// POUs/IO/AnalogInELMSingleSampleDINT
// AnalogIn FB to read and scale a single DINT (24bit) sample input from ELMxxxx terminal
// Set bit 3 (Options.3) to true to enable scaling based on +/-7812500 instead of legacy range values +/-838860x
FUNCTION_BLOCK AnalogInELMSingleSampleDINT EXTENDS AnalogInELMBase
VAR_INPUT
	Offset													:	LREAL := 0.0;

END_VAR                 									
VAR                                     	            	
END_VAR                                 	            	
VAR_OUTPUT                              	            	                                       	
	Q														:	LREAL;	//scaled result value
	In											AT  %I* 	: 	DINT; 	//Hardware Input 
END_VAR                                 	
VAR                                   	
END_VAR

(* Read single DINT sample value from ELM terminal and scale to user units									*)
(************************************************************************************************************)

(* evaluate statusword **************************************************************************************)
	SUPER^();
	
(* Scaling ******************************************************************)
	IF MaxValue <> MinValue 
	THEN	
		IF NOT Options.3
		THEN
			Q 	 											:= Offset + Scale(TO_LREAL(In) , -8388608.0, 8388607.0, MinValue , MaxValue);
		ELSE
			Q 	 											:= Offset + Scale(TO_LREAL(In), -7812500.0, 7812500.0, MinValue , MaxValue);
		END_IF	
		IF NoOfDigits > 0
		THEN
			Q												:= TO_FMLREAL(Q,NoOfDigits);
		END_IF
	
	ELSIF NoOfDigits > 0 (* Bsp PT100 *)
	THEN
		Q													:= Offset + TO_FMLREAL(In,NoOfDigits);
		
	ELSE  													
		Q 													:= 0.0;
	END_IF

	IF 	Error AND OutOnError <> 0.000000000000000001
	THEN
		Q													:= OutOnError;
	END_IF
(**********************************************************************************************************************)

METHOD FB_init : BOOL
VAR_INPUT
	bInitRetains : BOOL; // if TRUE, the retain variables are initialized (warm start / cold start)
	bInCopyCode : BOOL;  // if TRUE, the instance afterwards gets moved into the copy code (online change)
END_VAR
IF NOT bInCopyCode THEN
	NoOfDigits 							:= 2;
END_IF
END_METHOD

PROPERTY PUBLIC optEnableScaleExtRangeMode : bool
GET
optEnableScaleExtRangeMode := Options.3;
END_GET
SET
Options.3 := optEnableScaleExtRangeMode;
END_SET
END_PROPERTY

END_FUNCTION_BLOCK

// POUs/IO/AnalogInELMSingleSampleREAL
// AnalogIn FB to read and scale a single REAL sample input from ELMxxxx terminal
// Set bit 3 (Options.3) to true to enable scaling based on +/-7812500 instead of legacy range values +/-838860x
// NoOfDigits per default set to 3... 
FUNCTION_BLOCK AnalogInELMSingleSampleREAL EXTENDS AnalogInELMBase
VAR_INPUT
	Offset													:	LREAL := 0.0;
END_VAR                 									
VAR                                     	            	
END_VAR                                 	            	
VAR_OUTPUT                              	            	                                       	
	Q														:	LREAL;	//scaled result value
	In											AT  %I* 	: 	REAL; 	//Hardware Input 
END_VAR                                 	
VAR                                     	
END_VAR

(* Read single REAL sample value from ELM terminal and scale to user units									*)
(************************************************************************************************************)

(* evaluate statusword **************************************************************************************)
	SUPER^();
	
(* Scaling ******************************************************************)
	IF MaxValue <> MinValue 
	THEN			
		IF NOT Options.3
		THEN
			Q 	 											:= Offset + Scale(TO_LREAL(In), -8388608.0, 8388607.0, MinValue , MaxValue);
		ELSE
			Q 	 											:= Offset + Scale(TO_LREAL(In),  -7812500.0, 7812500.0, MinValue , MaxValue);		
		END_IF	
		
		IF NoOfDigits > 0
		THEN
			Q												:= TO_FMLREAL(Q,NoOfDigits);
		END_IF
	
	ELSIF NoOfDigits > 0 (* Bsp PT100 *)
	THEN
		Q													:= Offset + TO_FMLREAL(In,NoOfDigits);
		
	ELSE  													
		Q 													:= 0.0;
	END_IF


(**********************************************************************************************************************)

METHOD FB_init : BOOL
VAR_INPUT
	bInitRetains : BOOL; // if TRUE, the retain variables are initialized (warm start / cold start)
	bInCopyCode : BOOL;  // if TRUE, the instance afterwards gets moved into the copy code (online change)
END_VAR
IF NOT bInCopyCode THEN
	NoOfDigits 							:= 3;
END_IF
END_METHOD

PROPERTY PUBLIC optEnableScaleExtRangeMode : bool
GET
optEnableScaleExtRangeMode := Options.3;
END_GET
SET
Options.3 := optEnableScaleExtRangeMode;
END_SET
END_PROPERTY

END_FUNCTION_BLOCK

// POUs/IO/BlowOffSensors
{attribute 'no_check'}
//FB generates a pulse "Pulse" time based signal on every bit at Q (DWORD) for a certain lenght
//The sequecne will starts based on the seletcted time of interval if Enable is TRUE
//The FB can be used to activate air blow valves on by one to clean sensors in a dusty environment
FUNCTION_BLOCK BlowOffSensors
VAR_INPUT
	Enable													:	BOOL;			//FB will be processed as long as enable is TRUE
	StartManual												:	BOOL;			//starts FB without interval
	Interval												:	TIME := T#60M; 	//Blow of autostart interval
	Lenght													:	TIME := T#4S; 	//Duration of pulsing
	Pulse													:	TIME := T#500MS; //On/Off pulse duration
END_VAR                 									
VAR_OUTPUT              									
	Aktiv													:	BOOL;			//Busy is TRUE at the rising edge of Enable and stays TRUE as long as the FB is performing any action.  
{attribute 'displaymode':='binary'}    
	Q														:	DWORD := 0;		//Each bit will be set and reset based on the settings one by one 
END_VAR                 									
VAR                     									
	state													:	INT := 0;
	i														:	SINT ;
	TON_Interval											:	TON;
	TON_Lenght		 										: 	TON;
	TOF_Pulse	 											:	TOF;
END_VAR

(* Abblastaktgenerator					*)
(***************************************)

(* Intervalzeit ***********************************************************************)
IF Enable 
THEN
	CASE state OF
	0:
		TON_Interval(IN := FALSE);
		state 												:= 10;
		i 													:= -1;

	1:
		Aktiv := FALSE;
		TON_Interval(IN := Interval <> T#0MS , PT := Interval);
		IF TON_Interval.Q
			OR StartManual
		THEN
			TON_Interval(IN := FALSE);
			
			state 											:= 10;
			Aktiv 											:= TRUE;
			i 												:= -1;
		END_IF

	10:
		i := i + 1;
		IF i > 31 THEN
			state 											:= 1;
		ELSE
			TON_Lenght(IN := FALSE);
			TOF_Pulse(IN := FALSE);
			
			Q		 										:= 0;
			state 											:= 11;
		END_IF                  							

	11:
		TON_Lenght(IN := TRUE, PT := Lenght);

		IF 	TON_Lenght.Q
			AND Q = 0
		THEN
			state 											:= 10;
		ELSE
			IF 	NOT TOF_Pulse.Q 
				AND Q <> 0 
			THEN
				TOF_Pulse(IN:=TRUE  , PT:= Pulse);
				Q		 									:= 0;
			ELSIF NOT TOF_Pulse.Q 
				AND Q = 0 
			THEN
				TOF_Pulse(IN:= TRUE , PT:= Pulse) ;
				Q		 									:= SETBIT32(Q,i);
			END_IF
			(* Work Timer *)
			TOF_Pulse(IN:=FALSE);
		END_IF

	END_CASE
ELSE
	Aktiv 													:= FALSE;
	state 													:= 0;
	Q														:= 0;
END_IF

(**********************************************************************************************************)

END_FUNCTION_BLOCK

// POUs/TimeHelper/Pulse
{attribute 'no_check'}
//Generates a pulse signal 
FUNCTION_BLOCK Pulse
VAR_INPUT
	IN														: BOOL; //Start pulse generator
	PT_ON													: TIME; //Time pulse on	
	PT_OFF													: TIME; //Time pulse off 
END_VAR             										
VAR_OUTPUT          										
	Q														: BOOL; 
	RT														: BOOL; 
	FT														: BOOL;
END_VAR             										
VAR                 	
	TON_PULSE												: TON;
END_VAR

	(* Pulse generator																*)
	(********************************************************************************)

(* Reset flag *)
RT := FT													:= FALSE;
(* logic *)
IF 	Q AND(TON_PULSE.Q OR NOT IN)
THEN
	TON_PULSE(IN:=FALSE  , PT:= PT_OFF);
	FT 														:= Q;
	Q 														:= FALSE;
ELSIF NOT Q AND TON_PULSE.Q
	OR_ELSE In AND NOT TON_PULSE.IN 
THEN
	RT 														:= NOT Q;
	TON_PULSE(IN:= FALSE , PT:= PT_ON) ;
	Q 														:= TRUE;
END_IF

//Run timer
TON_PULSE(IN:=IN);

(***********************************************************************************************************************)

END_FUNCTION_BLOCK

// POUs/IO/Button
{attribute 'no_check'}
FUNCTION_BLOCK Button 
VAR_INPUT
	Enable													:	BOOL := TRUE;	//FB will be processed as long as enable is TRUE 
	RstTGL													:	BOOL := FALSE; 	//resets the Toggle signal
	SetTGL													:	BOOL := FALSE;	//sets the Toggle signal
	Force													:	BOOL := FALSE; 	//simulates Input signal
	Invert													:	BOOL := FALSE; 	//inverts the Hardware Input
	LED												AT  %Q*	:	BOOL;			//LED/Light hardware output
END_VAR         									
VAR_OUTPUT
	Q														:	BOOL;	//direct signal
	Q_RT													:	BOOL;	//R_Trig signal of delay Q
	Q_FT													:	BOOL;	//F_Trig signal of delay Q
	Q_TGL													:	BOOL;	//Toggle -> use flag Q_RT
	In												AT  %I*	:	BOOL; 	//Hardware Input
END_VAR
VAR
	Mem														:	BOOL;
END_VAR

(* Taster mit Togglefunktion V1.0						*)
(********************************************************)

(********************************************************)
Mem															:= Q;
Q 															:= ((In OR Force) XOR Invert) AND Enable;
Q_RT 														:= NOT Mem AND Q;
Q_FT														:= Mem AND NOT Q;
Q_TGL 														:= (Q_RT XOR Q_TGL);
(********************************************************)

METHOD PUBLIC setDisable : BOOL
VAR_INPUT
END_VAR
Enable 														:= FALSE;
setDisable													:= TRUE;
END_METHOD

METHOD PUBLIC setEnable : bool
VAR_INPUT
END_VAR
Enable 														:= TRUE;
setEnable													:= TRUE;
END_METHOD

METHOD PUBLIC setLedOFF : bool
VAR_INPUT
END_VAR
LED 														:= FALSE;
setLEDOff													:= TRUE;
END_METHOD

METHOD PUBLIC setLedON : booL
VAR_INPUT
END_VAR
LED 														:= TRUE;
setLedON													:= TRUE;
END_METHOD

METHOD PUBLIC TGL : booL //Return value = Q_TGL status
VAR_INPUT
END_VAR
TGL := Q_TGL 														:= NOT Q_TGL;
END_METHOD

METHOD PUBLIC TglOff : booL
VAR_INPUT
END_VAR
Q_TGL 														:= FALSE;
TglOFF														:= TRUE;
END_METHOD

METHOD PUBLIC TglOn : bool
VAR_INPUT
END_VAR
Q_TGL 														:= TRUE;
TglON														:= TRUE;
END_METHOD

END_FUNCTION_BLOCK

// POUs/IO/ButtonExt
{attribute 'no_check'}
//Button with delay function 
FUNCTION_BLOCK ButtonExt EXTENDS Button
VAR_INPUT
	PT_ON													:	TIME := T#0MS; 	//Delay for Q, Q_RT (TGL) and Q_FT
END_VAR
VAR_OUTPUT
	Q_DIRECT												:	BOOL; 	//Direct signal - undelayed
END_VAR
VAR
	TON														:	TON;
END_VAR

(* Button with toggle-function and on-delay		V1.5	*)
(********************************************************)

(********************************************************)
TON(IN := ((In OR Force) XOR Invert) AND Enable, PT := PT_ON);
Q_DIRECT 													:= TON.IN;
IF NOT Q    												
THEN        												
	Q 														:= TON.Q;
	Q_RT 													:= Q;
	Q_FT 													:= FALSE;
ELSE        												
	Q 														:= TON.IN;
	Q_RT 													:= FALSE;
	Q_FT 													:= NOT Q;
END_IF      	

Q_TGL := NOT RstTGL AND (Q_RT XOR Q_TGL OR SetTGL) ;

(********************************************************)

END_FUNCTION_BLOCK

// POUs/IO/InOut
{attribute 'no_check'}
FUNCTION_BLOCK InOut 
VAR_INPUT
	Q												AT  %Q*	:	BOOL; //Link to hardware output
END_VAR             								
VAR_OUTPUT          								
	In												AT  %I*	:	BOOL; //Link to hardware input
END_VAR
VAR
END_VAR

;

END_FUNCTION_BLOCK

// POUs/IO/InOutExt
{attribute 'no_check'}
FUNCTION_BLOCK InOutExt EXTENDS InOut IMPLEMENTS I_ActuatorOnOff
VAR_INPUT
	ResetTrig												:	BOOL;	//Resets error with rising edge
	Invert													:	BOOL ;			//Inverts the logic of varibale In (AT  %I*)
	PT_Timeout												:	TIME := T#3S;  	//Time value until Timeout of process (Error)
END_VAR                     				
VAR_OUTPUT                  				
	Busy													:	BOOL;			//Busy is TRUE at the rising edge of Execute and FALSE when one of the outputs Done, Aborted, or Error is set 
	ErrorOn													:	BOOL;			//Timeout error waiting for IN changing to TRUE
	ErrorOff												:	BOOL;			//Timeout error waiting for IN changing to FALSE
	Done													:	BOOL;			//The Done output is set when the commanded action has been completed successfully 
	Status													:	BYTE;			//8 different query Options (conditions see below)
END_VAR                     	
VAR                         	
	tonRM													:	ton;			
END_VAR

(* Actuator with feedback								*)
(********************************************************)

(********************************************************)
	IF Q 
	THEN
		SwitchOn();
	ELSE
		SwitchOff();
	END_IF
	_runtimeChk();
	_writeStatus();

(********************************************************)

METHOD PROTECTED _runtimeChk : BOOL
VAR_INPUT
END_VAR
	tonRM(
		IN	:= Busy AND NOT ResetTrig,  
		PT 	:= PT_Timeout,
		Q	=> );
		
	ErrorOff 												:= tonRM.Q AND NOT Q;
	ErrorOn 												:= tonRM.Q AND Q;

	_runtimeChk									:= TRUE;
END_METHOD

METHOD PROTECTED _writeStatus : BOOL
VAR_INPUT
END_VAR
	Status.0 												:= NOT Q;
	Status.1 												:= Q;
	Status.2 												:= NOT (In XOR Invert);
	Status.3 												:= In XOR Invert;
	Status.4 												:= NOT ErrorOff;
	Status.5 												:= NOT ErrorOn;
	Status.6 												:= NOT Status.7;
	Status.7 												:= ErrorOff OR ErrorOn;
	
	(* Result *)
	_writeStatus											:= TRUE;
END_METHOD

METHOD PUBLIC enable : BOOL //Result value = TRUE if successful executed (
VAR_INPUT 
	IN								: BOOL; //TRUE = ON/FALSE = OFF	
END_VAR
IF IN
THEN
	enable							:= switchOn();
ELSE
	enable							:= switchOff();
END_IF
END_METHOD

{attribute 'monitoring' := 'call'}
PROPERTY public inError : BOOL
GET
inError := ErrorON or ErrorOff;
END_GET
END_PROPERTY

{attribute 'monitoring' := 'call'}
PROPERTY public isBusy : bool
GET
isBusy := Busy;
END_GET
END_PROPERTY

{attribute 'monitoring' := 'call'}
PROPERTY public isOff : BOOL
GET
isOff := not Q;
END_GET
END_PROPERTY

{attribute 'monitoring' := 'call'}
PROPERTY public isOn : BOOL
GET
isOn := Q;
END_GET
END_PROPERTY

{attribute 'monitoring' := 'call'}
PROPERTY Public noFeed : BOOL
GET
noFeed := FALSE;
END_GET
END_PROPERTY

{attribute 'monitoring' := 'call'}
PROPERTY Public ok : bool
GET
ok := Q and Done or not Q and not Done;
END_GET
END_PROPERTY

METHOD PUBLIC reset : Bool
VAR_INPUT
END_VAR
tonRM(IN := FALSE);
reset := TRUE;
END_METHOD

METHOD public switchOff : BOOL
VAR_INPUT
END_VAR
	
	Q														:= FALSE;
	Done													:= NOT (In XOR Invert);
	Busy													:= NOT Done;
	switchOff												:= Done;
END_METHOD

METHOD public switchOn : BOOL
VAR_INPUT
END_VAR
	Q														:= TRUE;
	Done													:= (In XOR Invert);
	Busy													:= NOT Done;
	switchOn												:= Done;
END_METHOD

END_FUNCTION_BLOCK

// POUs/IpcDiag/MDP/InfoModuls/MDP_CPU
{attribute 'no_check'}
//Wrapper for available MDP_xxxx FBs of the lib, based on Beckhoff MDP - invalid values are reported via EventLogger 
//based on Tc2_MDP.lib - please see Beckhoff documentation for further information about Tc2_MDP.lib (IPC diagnostics)
FUNCTION_BLOCK MDP_CPU  EXTENDS FbBase
VAR_OUTPUT CONSTANT
	MIN_CPU													:	INT := 1;
	MAX_CPU													:	INT := 8;
END_VAR                 									
VAR_INPUT               									
	AmsNetId												: 	T_AmsNetId := '';				//AmsNetId as text
	Timeout													:	TIME := DEFAULT_ADS_TIMEOUT;	//Ads timeout
END_VAR                 									
VAR_OUTPUT              									
	Frequency												:  ARRAY[MIN_CPU..MAX_CPU] OF	UDINT;	//current CPU frequency
	Usage													:	ARRAY[MIN_CPU..MAX_CPU] OF	UINT;	//current CPU usage in %
	Temperature												:	ARRAY[MIN_CPU..MAX_CPU] OF	INT;	//current CPU temperature in °C
	AverageFrequency 										:	UDINT;		//average CPU frequency
	AverageUsage	 										:	UINT;		//average CPU usage in %
	AverageTemperature										:	INT;		//average CPU temperature in °C
	Count													:	INT; 		//number of CPUs
	ErrorGrp												:	E_MDP_ErrGroup := eMDP_Err_NoError;
END_VAR
VAR
	idx														:	INT := 1;
	MDP_ScanModules											:	FB_MDP_ScanModules := ( nModuleType 	:= eMDP_ModT_CPU , iModIdx		:= 0);
	MDP_Read												: 	FB_MDP_ReadModuleContent;
	SplitErrorId											:	FB_MDP_SplitErrorID;
	DstBuf													:	ARRAY[0..13] OF BYTE;
END_VAR

(* Read CPU Information 						V1.0		*)
(************************************************************)

(* Start Read ***********************************************)
	IF Execute
		AND state = 0
	THEN
		MEMSET(ADR(Frequency),0,SIZEOF(Frequency));
		MEMSET(ADR(Usage),0,SIZEOF(Usage));
		MEMSET(ADR(Temperature),0,SIZEOF(Temperature));
		AverageFrequency									:= 0;
		AverageUsage										:= 0;
		AverageTemperature									:= 0;
		Count												:= 0;
		Busy												:= TRUE;
		Done												:= FALSE;
		Error												:= FALSE;
		ErrorId												:= 0;
		ErrorGrp											:= eMDP_Err_NoError;
		MDP_Read(bExecute := FALSE);
		MDP_ScanModules(
			bExecute		:= FALSE,
			nModuleType		:= eMDP_ModT_CPU,
			iModIdx			:= 0,
			tTimeout		:= timeout,
			sAmsNetId		:= AmsNetId,
			bBusy			=> ,
			bError			=> ,
			nErrID			=> ,
			nDynModuleId	=> ,
			iModuleTypeCount=> ,
			iModuleCount	=> );
			
		MDP_ScanModules(bExecute		:= TRUE);		
		state												:= 1 ;
		
	ELSIF NOT Execute
		AND State = 99
	THEN
		state												:= 0;
		Busy												:= FALSE;
		Done												:= FALSE;
		Error												:= FALSE;
		ErrorId												:= 0;
		ErrorGrp											:= eMDP_Err_NoError;
	END_IF


	CASE state OF
	0:
		;
	1:
		MDP_ScanModules();
		IF NOT MDP_ScanModules.bBusy
		THEN
			IF MDP_ScanModules.bError
			THEN
				Busy										:= FALSE;
				Error										:= TRUE;
				SplitErrorId(
					nErrID		:= MDP_ScanModules.nErrID,
					eErrGroup	=> ErrorGrp ,
					nErrCode	=> ErrorId);
				state										:= 99;
				MDP_ScanModules(bExecute := FALSE);
			ELSE
				Count										:= MDP_ScanModules.iModuleTypeCount;
				MDP_Read.stMDP_DynAddr.nArea				:= 16#8;
				MDP_Read.stMDP_DynAddr.nModuleId			:= MDP_ScanModules.nDynModuleId;
				MDP_Read.stMDP_DynAddr.nSubIdx				:= 0;
				MDP_Read.stMDP_DynAddr.nTableId				:= 1;
				MDP_Read(bExecute := FALSE);
				idx											:= 1;
				IF Count = 0
				THEN
					Busy									:= FALSE;
					Error									:= TRUE;
					ErrorId									:= MDP_Read.nErrID;
					state									:= 99;
				ELSE
					MDP_Read(
						bExecute		:= TRUE,
						stMDP_DynAddr	:= ,
						iSubIdxCount	:= 4,
						pDstBuf			:= ADR(DstBuf),
						cbDstBufLen		:= SIZEOF(DstBuf),
						tTimeout		:= timeout,
						sAmsNetId		:= AmsNetId,
						bBusy			=> ,
						bError			=> ,
						nErrID			=> ,
						iErrPos			=> ,
						arrStartIdx		=> );
					state									:= 2;
				END_IF
			END_IF

		END_IF

	2:
		MDP_Read( pDstBuf := ADR(DstBuf), cbDstBufLen := SIZEOF(DstBuf));
		
		IF NOT MDP_Read.bBusy
		THEN
			IF MDP_Read.bError AND MDP_Read.iErrPos <> 4 AND MDP_Read.bExecute
			THEN
				Busy										:= FALSE;
				Error										:= TRUE;
				SplitErrorId(
					nErrID		:= MDP_Read.nErrID,
					eErrGroup	=> ErrorGrp ,
					nErrCode	=> ErrorId);
				state										:= 99;
				MDP_Read(bExecute := FALSE);
			ELSE
				(* copy freq *)
				IF MDP_Read.arrStartIdx[1] >= 0
				THEN
					MEMCPY( ADR(Frequency[idx]) , ADR(DstBuf[MDP_Read.arrStartIdx[1]]) , SIZEOF(Frequency[idx]) );
				END_IF
				(* copy usage *)
				IF MDP_Read.arrStartIdx[2] <> 0
				THEN
					MEMCPY(ADR(Usage[idx]) , ADR(DstBuf[MDP_Read.arrStartIdx[2]]) , SIZEOF(Usage[idx]) );
				END_IF
				(* copy temp in availible *)
				IF MDP_Read.arrStartIdx[3] <> 0
				THEN
					MEMCPY(ADR(Temperature[idx]) , ADR(DstBuf[MDP_Read.arrStartIdx[3]]) , SIZEOF(Temperature[idx]) ) ;
				END_IF

				MDP_Read(bExecute := FALSE);
				MDP_Read.stMDP_DynAddr.nModuleId := MDP_Read.stMDP_DynAddr.nModuleId + 1;
				
				idx 										:= idx + 1;
				IF idx > Count AND Count > 0
				THEN
					FOR idx := 1 TO Count
					DO
						AverageFrequency 					:= AverageFrequency + Frequency[idx];
						AverageUsage 						:= AverageUsage + Usage[idx];
						AverageTemperature 					:= AverageTemperature + Temperature[idx];
					END_FOR                         		
                                                    		
					AverageFrequency						:= AverageFrequency / INT_TO_UDINT(Count);
					AverageUsage							:= AverageUsage / INT_TO_UINT(Count);
					AverageTemperature						:=	AverageTemperature / INT_TO_SINT(Count);
                                                        	
					Busy									:= FALSE;
					Done									:= TRUE;
					state									:= 99;
				ELSE
					MDP_Read(bExecute := TRUE);
				END_IF
			END_IF
		END_IF

	99: ;

	ELSE
		;
	END_CASE

	(* reset state for next start *)
	IF NOT Execute
		AND state = 99
	THEN
		state												:= 0;
	END_IF

(****************************************************************************************************)

END_FUNCTION_BLOCK

// POUs/IpcDiag/MDP/InfoModuls/MDP_Fan
{attribute 'no_check'}
FUNCTION_BLOCK MDP_Fan EXTENDS FbBase
VAR_OUTPUT CONSTANT
	MIN_FAN													:	INT := 1;
	MAX_FAN													:	INT := 4;
END_VAR                     								
VAR_INPUT                   								
	AmsNetId												: 	T_AmsNetId := '';					//AmsNetId as text
	Timeout													:	TIME := DEFAULT_ADS_TIMEOUT;		//Ads timeout
END_VAR                     								
VAR_OUTPUT                  								
	Speed													:  ARRAY[MIN_FAN..MAX_FAN] OF	INT;	//current fan speed
	Count													:	INT; 	//number of CPUs
	ErrorGrp												:	E_MDP_ErrGroup := eMDP_Err_NoError;
END_VAR                     								
VAR                         								
	idx														:	INT := 1;
	MDP_ScanModules											:	FB_MDP_ScanModules := ( nModuleType 	:= eMDP_ModT_FAN , iModIdx		:= 0);
	MDP_Read												: 	FB_MDP_Read;
	SplitErrorId											:	FB_MDP_SplitErrorID;
	DstBuf													:	ARRAY[0..4] OF BYTE;
END_VAR

(* Read FAN Information 					V1.0	*)
(****************************************************)

(* Start Read *******************************************************)
	IF Execute
		AND state = 0
	THEN
		MEMSET(ADR(Speed),0,SIZEOF(Speed));
		Count												:= 0;
		Busy												:= TRUE;
		Done												:= FALSE;
		Error												:= FALSE;
		ErrorId												:= 0;
		ErrorGrp											:= eMDP_Err_NoError;
		MDP_Read(bExecute := FALSE);
		MDP_ScanModules(
			bExecute		:= FALSE,
			nModuleType		:= eMDP_ModT_FAN,
			iModIdx			:= 0,
			tTimeout		:= timeout,
			sAmsNetId		:= AmsNetId,
			bBusy			=> ,
			bError			=> ,
			nErrID			=> ,
			nDynModuleId	=> ,
			iModuleTypeCount=> ,
			iModuleCount	=> );
			
		MDP_ScanModules(bExecute		:= TRUE);		
		state												:= 1;
		
	ELSIF NOT Execute
		AND State = 99
	THEN
		state												:= 0;
		Busy												:= FALSE;
		Done												:= FALSE;
		Error												:= FALSE;
		ErrorId												:= 0;
		ErrorGrp											:= eMDP_Err_NoError;
	END_IF


	CASE state OF
	0:
		;

	1:
		MDP_ScanModules();
		IF NOT MDP_ScanModules.bBusy
		THEN
			IF MDP_ScanModules.bError
			THEN
				Busy										:= FALSE;
				Error										:= TRUE;
				SplitErrorId(
					nErrID		:= MDP_ScanModules.nErrID,
					eErrGroup	=> ErrorGrp ,
					nErrCode		=> ErrorId);
				state										:= 99;
				MDP_ScanModules(bExecute := FALSE);
			ELSE
				Count										:= MDP_ScanModules.iModuleTypeCount;
				MDP_Read(bExecute := FALSE);
				MDP_Read.stMDP_DynAddr.nArea				:= 16#8;
				MDP_Read.stMDP_DynAddr.nModuleId			:= MDP_ScanModules.nDynModuleId;
				MDP_Read.stMDP_DynAddr.nTableId				:= 1;
				MDP_Read.stMDP_DynAddr.nSubIdx				:= 1;
				
				MDP_Read(
					stMDP_DynAddr	:= ,		(* address to request subindex Count of AdressList *)
					pDstBuf			:= ADR(DstBuf),
					cbDstBufLen		:= SIZEOF(DstBuf),
					bExecute		:= TRUE,
					tTimeout		:= Timeout,
					sAmsNetId		:= AmsNetId,
					bBusy			=> ,
					bError			=> ,
					nErrId			=> );
				idx											:= 1;
				state										:= 2;
			END_IF

		END_IF

	2:
		MDP_Read( pDstBuf	:= ADR(DstBuf), cbDstBufLen := SIZEOF(DstBuf));
		IF NOT MDP_Read.bBusy
		THEN
			IF MDP_Read.bError AND MDP_Read.bExecute
			THEN
				Busy										:= FALSE;
				Error										:= TRUE;
				SplitErrorId(
					nErrID		:= MDP_Read.nErrID,
					eErrGroup	=> ErrorGrp ,
					nErrCode	=> ErrorId);
				state										:= 99;
				MDP_Read(bExecute := FALSE);
			ELSE
				MDP_Read(bExecute := FALSE);
				MEMCPY(ADR(Speed[idx]), ADR(DstBuf), SIZEOF(Speed[idx]));
				IF idx < Count
				THEN
					MDP_Read.stMDP_DynAddr.nModuleId		:= MDP_Read.stMDP_DynAddr.nModuleId + 1;
					idx 									:= idx + 1;
				ELSE                                    	
					Busy									:= FALSE;
					Done									:= TRUE;
					state									:= 99;
				END_IF

				MDP_Read(
					stMDP_DynAddr	:= ,(* address to request subindex Count of AdressList *)
					pDstBuf			:= ADR(DstBuf),
					cbDstBufLen		:= SIZEOF(DstBuf),
					bExecute		:= NOT MDP_Read.bBusy AND state = 2,
					tTimeout		:= Timeout,
					sAmsNetId		:= AmsNetId,
					bBusy			=> ,
					bError			=> ,
					nErrId			=> );
			END_IF
		END_IF

	99: ;

	ELSE
		;
	END_CASE


	(* reset state for next start *)
	IF NOT Execute
		AND state = 99
	THEN
		state												:= 0;
	END_IF

(****************************************************************************************************)

END_FUNCTION_BLOCK

// POUs/IpcDiag/MDP/InfoModuls/MDP_Mainboard
{attribute 'no_check'}
FUNCTION_BLOCK MDP_Mainboard  EXTENDS FbBase
VAR_OUTPUT CONSTANT
	MIN_VOLTAGE												:	INT := 1;
	MAX_VOLTAGE												:	INT := 20;

(* Voltage Location *)
 	VLOC_UNKNOWN											:	INT := 0;
	VLOC_OTHER												:	INT := 1;
 	VLOC_PROCESSOR											:	INT := 2;
 	VLOC_DISK												:	INT := 3;
 	VLOC_SYSTEM_MANAGEMENT_MODULE							:	INT := 4;
 	VLOC_MOTHERBOARD										:	INT := 5;
 	VLOC_MEMORY_MODULE										:	INT := 6;
 	VLOC_POWER_SUPPLY										:	INT := 7;
 	VLOC_ADDIN_CARD											:	INT := 8;
 	VLOC_FRONT_PANEL_BOARD									:	INT := 9;
 	VLOC_BACK_PANEL_BOARD									:	INT := 10;
 	VLOC_PERIPHERIE											:	INT := 11;
 	VLOC_CHASSIS											:	INT := 12;
 	VLOC_BATTERY											:	INT := 13;
 	VLOC_UPS												:	INT := 14;
	VLOC_GRAFFIC_BOARD										:	INT := 15;
 	VLOC_SUPERIO											:	INT := 16;
	VLOC_CHIPSET											:	INT := 17;
END_VAR                             						
VAR_INPUT                           						
	AmsNetId												: 	T_AmsNetId := '';				//AmsNetId as text
	Timeout													:	TIME := DEFAULT_ADS_TIMEOUT;	//Ads timeout
END_VAR
VAR_OUTPUT
	MB_Type													:	STRING(20);	//Type of Mainboard
	SerielNo												:	STRING(20);	//Serial number of Mainboard
	ProdDate												:	STRING(20);	//Production date of Mainboard
	BootCount												:	UDINT;		//total number of boots
	OpTime													:	UDINT; 		//Operating Time
	MinBoardTemp											:	DINT;		//minimum board temperature
	MaxBoardTemp											:	DINT;		//maximum board temperature
	MinInputVolt											:	DINT;		//minimum board input voltage
	MaxInputVolt											:	DINT;		//maximum board input voltage
	MB_Temp													:	INT;		//current board temperature
	IPC_SerielNo											:	STRING(20);	//industrial PC serial number
                        									
	VoltLocation											:  	ARRAY[MIN_VOLTAGE..MAX_VOLTAGE] OF INT;	//voltage location
	VoltageValue											:	ARRAY[MIN_VOLTAGE..MAX_VOLTAGE] OF INT;	//voltage value
	VoltageNominal											:	ARRAY[MIN_VOLTAGE..MAX_VOLTAGE] OF INT;	//nominal voltage
	VoltCount												:	INT; 		//number of measuring points
	ErrorGrp												:	E_MDP_ErrGroup := eMDP_Err_NoError;

END_VAR                 									
VAR                     									
	idx														:	INT := 1;
	MDP_ScanModules											:	FB_MDP_ScanModules := ( nModuleType 	:= eMDP_ModT_Mainboard , iModIdx		:= 0);
	MDP_Read												: 	FB_MDP_Read;
	SplitErrorId											:	FB_MDP_SplitErrorID;
	DstBuf													:	ARRAY[0..21] OF BYTE;
END_VAR

(* Read Mainboard Information 				V1.0	*)
(****************************************************)

(* Start Read *******************************************************)
	IF Execute
		AND state = 0
	THEN
		MB_Type												:= '';
		SerielNo											:= '';
		ProdDate											:= '';
		BootCount											:= 0;
		OpTime												:= 0;
		MinBoardTemp										:= 0;
		MaxBoardTemp										:= 0;
		MinInputVolt										:= 0;
		MaxInputVolt										:= 0;
		MB_Temp												:= 0;
		MEMSET(ADR(VoltLocation),0,SIZEOF(VoltLocation));
		MEMSET(ADR(VoltageValue),0,SIZEOF(VoltageValue));
		MEMSET(ADR(VoltageNominal),0,SIZEOF(VoltageNominal));
		VoltCount											:= 0;

		Busy												:= TRUE;
		Done												:= FALSE;
		Error												:= FALSE;
		ErrorId												:= 0;
		ErrorGrp											:= eMDP_Err_NoError;
		MDP_Read(bExecute := FALSE);
		MDP_ScanModules(
			bExecute			:= FALSE,
			nModuleType			:= eMDP_ModT_Mainboard,
			iModIdx				:= 0,
			tTimeout			:= timeout,
			sAmsNetId			:= AmsNetId,
			bBusy				=> ,
			bError				=> ,
			nErrID				=> ,
			nDynModuleId		=> ,
			iModuleTypeCount	=> ,
			iModuleCount		=> );

		MDP_ScanModules(bExecute:= TRUE);	
		state												:= 1;
		
	ELSIF NOT Execute
		AND State = 99
	THEN
		state												:= 0;
		Busy												:= FALSE;
		Done												:= FALSE;
		Error												:= FALSE;
		ErrorId												:= 0;
		ErrorGrp											:= eMDP_Err_NoError;
	END_IF


	CASE state OF
	0:
		;

	1:
		MDP_ScanModules();
		IF NOT MDP_ScanModules.bBusy
		THEN
			IF MDP_ScanModules.bError
			THEN
				Busy										:= FALSE;
				Error										:= TRUE;
				SplitErrorId(
					nErrID		:= MDP_ScanModules.nErrID,
					eErrGroup	=> ErrorGrp ,
					nErrCode	=> ErrorId);
				state										:= 99;
				MDP_ScanModules(bExecute := FALSE);
			ELSE
				MDP_Read(bExecute := FALSE);
				MDP_Read.stMDP_DynAddr.nArea				:= 16#8;
				MDP_Read.stMDP_DynAddr.nModuleId			:= MDP_ScanModules.nDynModuleId;
				MDP_Read.stMDP_DynAddr.nTableId				:= 1;
				MDP_Read.stMDP_DynAddr.nSubIdx				:= 0;
				idx											:= 1;
				state										:= 2;
			END_IF                                  		

		END_IF

	2:
		MDP_Read( pDstBuf	:= ADR(DstBuf), cbDstBufLen := SIZEOF(DstBuf));
		IF NOT MDP_Read.bBusy
		THEN
			IF MDP_Read.bError AND MDP_Read.bExecute
			THEN
				Busy										:= FALSE;
				Error										:= TRUE;
				SplitErrorId(
					nErrID		:= MDP_Read.nErrID,
					eErrGroup	=> ErrorGrp ,
					nErrCode	=> ErrorId);
				state										:= 99;
				MDP_Read(bExecute := FALSE);
			ELSE
				MDP_Read(bExecute := FALSE);
				CASE MDP_Read.stMDP_DynAddr.nTableId OF
				1:
					CASE MDP_Read.stMDP_DynAddr.nSubIdx OF
					0:
						MDP_Read.stMDP_DynAddr.nSubIdx		:= 1;

					1:
						MEMCPY(ADR(MB_Type), ADR(DstBuf), MIN(MDP_Read.nCount, SIZEOF(MB_Type)) );
						MDP_Read.stMDP_DynAddr.nSubIdx		:= 2;

					2:
						MEMCPY(ADR(SerielNo), ADR(DstBuf), MIN(MDP_Read.nCount, SIZEOF(SerielNo)) );
						MDP_Read.stMDP_DynAddr.nSubIdx		:= 3;

					3:
						MEMCPY(ADR(ProdDate), ADR(DstBuf), MIN(MDP_Read.nCount, SIZEOF(ProdDate)) );
						MDP_Read.stMDP_DynAddr.nSubIdx		:= 4;

					4:
						MEMCPY(ADR(BootCount), ADR(DstBuf), SIZEOF(BootCount));
						MDP_Read.stMDP_DynAddr.nSubIdx		:= 5;

					5:
						MEMCPY(ADR(OpTime), ADR(DstBuf), SIZEOF(OpTime));
						MDP_Read.stMDP_DynAddr.nSubIdx		:= 6;

					6:
						MEMCPY(ADR(MinBoardTemp), ADR(DstBuf), SIZEOF(MinBoardTemp));
						MDP_Read.stMDP_DynAddr.nSubIdx		:= 7;

					7:
						MEMCPY(ADR(MaxBoardTemp), ADR(DstBuf), SIZEOF(MaxBoardTemp));
						MDP_Read.stMDP_DynAddr.nSubIdx		:= 8;

					8:
						MEMCPY(ADR(MinInputVolt), ADR(DstBuf), SIZEOF(MinInputVolt));
						MDP_Read.stMDP_DynAddr.nSubIdx		:= 9;

					9:
						MEMCPY(ADR(MaxInputVolt), ADR(DstBuf), SIZEOF(MaxInputVolt));
						MDP_Read.stMDP_DynAddr.nSubIdx		:= 10;

					10:
						MEMCPY(ADR(MB_Temp), ADR(DstBuf), SIZEOF(MB_Temp));
						MDP_Read.stMDP_DynAddr.nSubIdx		:= 0;
						MDP_Read.stMDP_DynAddr.nTableId		:= 4;
					END_CASE

				4:
					CASE MDP_Read.stMDP_DynAddr.nSubIdx OF
					0:
						MEMCPY(ADR(VoltCount), ADR(DstBuf), SIZEOF(VoltCount) );
						IF VoltCount > 0 THEN
							MDP_Read.stMDP_DynAddr.nSubIdx	:= 1;
						ELSE						
							state							:= 3;
						END_IF

					1..255:
						MEMCPY(ADR(VoltLocation[MDP_Read.stMDP_DynAddr.nSubIdx]), ADR(DstBuf), SIZEOF(VoltLocation[MIN_VOLTAGE]));
						MDP_Read.stMDP_DynAddr.nSubIdx	:= MDP_Read.stMDP_DynAddr.nSubIdx + 1;
						
						IF MDP_Read.stMDP_DynAddr.nSubIdx > VoltCount
						THEN
							MDP_Read.stMDP_DynAddr.nSubIdx	:= 1;
							MDP_Read.stMDP_DynAddr.nTableId	:= 5;
						END_IF
					END_CASE

				5:
					CASE MDP_Read.stMDP_DynAddr.nSubIdx OF
					1..255:
						MEMCPY(ADR(VoltageValue[MDP_Read.stMDP_DynAddr.nSubIdx]), ADR(DstBuf), SIZEOF(VoltageValue[MIN_VOLTAGE]));
						MDP_Read.stMDP_DynAddr.nSubIdx	:= MDP_Read.stMDP_DynAddr.nSubIdx + 1;
						
						IF MDP_Read.stMDP_DynAddr.nSubIdx > VoltCount
						THEN
							MDP_Read.stMDP_DynAddr.nSubIdx	:= 1;
							MDP_Read.stMDP_DynAddr.nTableId	:= 6;
						END_IF
					END_CASE

				6:
					CASE MDP_Read.stMDP_DynAddr.nSubIdx OF
					1..255:
						MEMCPY(ADR(VoltageNominal[MDP_Read.stMDP_DynAddr.nSubIdx]), ADR(DstBuf), SIZEOF(VoltageNominal[MIN_VOLTAGE]));
						MDP_Read.stMDP_DynAddr.nSubIdx	:= MDP_Read.stMDP_DynAddr.nSubIdx + 1;
						
						IF MDP_Read.stMDP_DynAddr.nSubIdx > VoltCount
						THEN
							state							:= 3;
						END_IF
					END_CASE
				END_CASE

				MDP_Read(
					stMDP_DynAddr	:= ,		(* address to request subindex Count of AdressList *)
					pDstBuf			:= ADR(DstBuf),
					cbDstBufLen		:= SIZEOF(DstBuf),
					bExecute		:= NOT MDP_Read.bBusy AND state = 2,
					tTimeout		:= Timeout,
					sAmsNetId		:= AmsNetId,
					bBusy			=> ,
					bError			=> ,
					nErrId			=> );
			END_IF
		END_IF

	3: //Start lesen der IPC Seriennummer 
		MDP_Read.stMDP_DynAddr.nArea						:= INT_TO_BYTE(eMDP_Area_DeviceArea);
		MDP_Read.stMDP_DynAddr.nModuleId					:= 16#9F;
		MDP_Read.stMDP_DynAddr.nTableId						:= 16#00;
		MDP_Read.stMDP_DynAddr.nSubIdx						:= 16#00;
		
		MDP_Read(
			stMDP_DynAddr	:= ,		(* address to request subindex Count of AdressList *)
			pDstBuf			:= ADR(IPC_SerielNo),
			cbDstBufLen		:= SIZEOF(IPC_SerielNo),
			bExecute		:= NOT MDP_Read.bBusy,
			tTimeout		:= Timeout,
			sAmsNetId		:= AmsNetId,
			bBusy			=> ,
			bError			=> ,
			nErrId			=> );	
			
		state												:= 4;	
	
	4:
		MDP_Read( pDstBuf	:= ADR(IPC_SerielNo), cbDstBufLen := SIZEOF(IPC_SerielNo));
		IF NOT MDP_Read.bBusy
		THEN
			IF MDP_Read.bError AND MDP_Read.bExecute
			THEN
				Busy										:= FALSE;
				Error										:= TRUE;
				SplitErrorId(
					nErrID		:= MDP_Read.nErrID,
					eErrGroup	=> ErrorGrp ,
					nErrCode	=> ErrorId);
				state										:= 99;	
			ELSE			                        		
				Busy										:= FALSE;
				Done										:= TRUE;
				state										:= 99;
			END_IF
			MDP_Read(bExecute := FALSE);
			
		END_IF

	99: ;

	ELSE
		;
	END_CASE


	(* reset state for next start *)
	IF NOT Execute
		AND state = 99
	THEN
		state												:= 0;
	END_IF

(****************************************************************************************************)

END_FUNCTION_BLOCK

// POUs/IpcDiag/MDP/InfoModuls/MDP_RaidSimple
{attribute 'no_check'}
FUNCTION_BLOCK MDP_RaidSimple  EXTENDS FbBase
VAR_OUTPUT CONSTANT
	MIN_DRIVE												:	INT := 1;
	MAX_DRIVE												:	INT := 4;
	                    									
//Cntr state            									
	CS_UNKNOWN												:	INT := 0;
	CS_GOOD													:	INT := 1;
	CS_FAILED												:	INT := 2; 
	CS_OFFLINE												:	INT := 3; 
	CS_POWER_OFF											:	INT := 4;
	                    									
//Cntr offline reason   									
	COR_NO_REASON											:	INT := 0;
	COR_INITIALIZING										:	INT := 1;
	COR_BUS_DEGRADED										:	INT := 2;
	COR_BUS_FAILURE											:	INT := 3;
	                    									
//Set state             									
	SS_OK													:	INT := 0;
	SS_DEGRADED												:	INT := 1;
	SS_REBUILDING											:	INT := 2;
	SS_FAILED												:	INT := 3;
	                    									
//Drive state		    									
	DS_OK													:	INT := 0;
	DS_REBUILDING											:	INT := 1;
	DS_FAILED 												:	INT := 2;
	DS_DEGRADED 											:	INT := 3;
END_VAR                 									
VAR_INPUT               									
	AmsNetId												: 	T_AmsNetId := '';	//AmsNetId as text
	Timeout													:	TIME := DEFAULT_ADS_TIMEOUT;	//Ads timeout
END_VAR                 									
VAR_OUTPUT              									
(* Raid Data *)         									
	CntrState												:	INT := CS_UNKNOWN;		//current controller state
	CntrOfflReason 											: 	INT := COR_NO_REASON;	//reason for controller offline
                        									
	SetType													:	USINT;					//type of RAID system
	SetState												:	INT := SS_OK;			
	SetInfo													:	USINT; (* 	If SetStatus = OK, THEN Info will be 0.
																					If SetStatus = DEGRADED, then Info will contain the failed drive index number.1
																					If SetStatus = REBUILDING, then Info will contain the percentage complete. The value will be in the range of 0 to 100 (0h to 64h).
																					If SetStatus == FAILED, then Info will be 0 or vendor specific. Since the failure modes could include drive or controller failures, Info may provide a vendor specific error code to indicate which component led to the failed status. *)
	CountDrives												:	UINT;
	DriveSTATE												:	ARRAY[MIN_DRIVE..MAX_DRIVE] OF INT; //current state of drive
	CountRAIDSets											:	UINT; 		//Count RAID sets
	ErrorGrp												:	E_MDP_ErrGroup := eMDP_Err_NoError;
END_VAR                 									
VAR                     									
	idx														:	INT := 1;
	MDP_ScanModules											:	FB_MDP_ScanModules := ( nModuleType 	:= eMDP_ModT_RAID , iModIdx		:= 0);
	MDP_Read												: 	FB_MDP_Read;
	SplitErrorId											:	FB_MDP_SplitErrorID ;
	DstBuf													:	ARRAY[0..4] OF BYTE;
END_VAR

(* Read RAID Information 						V1.0	*)
(* only for RAID set 1									*)
(* not more then MAX_DRIVES per RAID set				*)
(********************************************************)

(* Start Read *******************************************)
	IF Execute
		AND state = 0
	THEN
		CntrState											:= CS_UNKNOWN;
		CntrOfflReason 										:= COR_NO_REASON;
		SetType												:= 0;
		SetState											:= SS_OK;
		SetInfo												:= 0;
		CountDrives											:= 0;
		MEMSET(ADR(DriveSTATE),0,SIZEOF(DriveSTATE));   	
		CountRAIDSets										:= 0;
                                                        	
		Busy												:= TRUE;
		Done												:= FALSE;
		Error												:= FALSE;
		ErrorId												:= 0;
		ErrorGrp											:= eMDP_Err_NoError;
		MDP_Read(bExecute := FALSE);
		MDP_ScanModules(
			bExecute		:= FALSE,
			nModuleType		:= eMDP_ModT_RAID,
			iModIdx			:= 0,
			tTimeout		:= timeout,
			sAmsNetId		:= AmsNetId,
			bBusy			=> ,
			bError			=> ,
			nErrID			=> ,
			nDynModuleId	=> ,
			iModuleTypeCount=> ,
			iModuleCount	=> );
			
		MDP_ScanModules(bExecute:= TRUE);
		state												:= 1;
	ELSIF NOT Execute
		AND State = 99
	THEN
		state												:= 0;
		Busy												:= FALSE;
		Done												:= FALSE;
		Error												:= FALSE;
		ErrorId												:= 0;
		ErrorGrp											:= eMDP_Err_NoError;
	END_IF


	CASE state OF
	0:
		;
	1:
		MDP_ScanModules();
		IF NOT MDP_ScanModules.bBusy
		THEN
			IF MDP_ScanModules.bError
			THEN
				Busy										:= FALSE;
				Error										:= TRUE;
				SplitErrorId(
					nErrID		:= MDP_ScanModules.nErrID,
					eErrGroup	=> ErrorGrp ,
					nErrCode	=> ErrorId);
				state										:= 99;
				MDP_ScanModules(bExecute := FALSE);
			ELSE
				MDP_Read(bExecute := FALSE);
				MDP_Read.stMDP_DynAddr.nArea				:= 16#8;
				MDP_Read.stMDP_DynAddr.nModuleId			:= MDP_ScanModules.nDynModuleId;
				MDP_Read.stMDP_DynAddr.nTableId				:= 16#1;
				MDP_Read.stMDP_DynAddr.nSubIdx				:= 0;
				state										:= 2;
			END_IF

		END_IF

	2:
		MDP_Read( pDstBuf	:= ADR(DstBuf), cbDstBufLen := SIZEOF(DstBuf));
		IF NOT MDP_Read.bBusy
		THEN
			IF MDP_Read.bError AND MDP_Read.bExecute
			THEN
				IF MDP_Read.stMDP_DynAddr.nTableId = 16#2
					AND MDP_Read.stMDP_DynAddr.nSubIdx = 1
				THEN (* No RaidSystem found *)
					Busy									:= FALSE;
					Done									:= TRUE;
					state									:= 99;
				ELSE
					Busy									:= FALSE;
					Error									:= TRUE;
					SplitErrorId(
						nErrID		:= MDP_Read.nErrID,
						eErrGroup	=> ErrorGrp ,
						nErrCode	=> ErrorId);
				END_IF
				state										:= 99;
				MDP_Read(bExecute := FALSE);
			ELSE
				MDP_Read(bExecute := FALSE);
				CASE MDP_Read.stMDP_DynAddr.nTableId OF
				16#1: (* Controller Info *)
					CASE MDP_Read.stMDP_DynAddr.nSubIdx	OF
					0:
						MDP_Read.stMDP_DynAddr.nSubIdx		:= 1;

					1:
						MEMCPY(ADR(CntrState), ADR(DstBuf), SIZEOF(CntrState));
						MDP_Read.stMDP_DynAddr.nSubIdx		:= 2;

					2:
						MEMCPY(ADR(CntrOfflReason), ADR(DstBuf), SIZEOF(CntrOfflReason));
						MDP_Read.stMDP_DynAddr.nSubIdx		:= 0;
						MDP_Read.stMDP_DynAddr.nTableId		:= 16#2;
					END_CASE

				16#2: (* Raid Sets Type *)
					CASE MDP_Read.stMDP_DynAddr.nSubIdx	OF
					0:
						MEMCPY(ADR(CountRAIDSets), ADR(DstBuf), SIZEOF(CountRAIDSets));
						MDP_Read.stMDP_DynAddr.nSubIdx		:= 1;

					1:
						MEMCPY(ADR(SetType), ADR(DstBuf), SIZEOF(SetType));
						MDP_Read.stMDP_DynAddr.nSubIdx		:= 1;
						MDP_Read.stMDP_DynAddr.nTableId		:= 16#3;
					END_CASE

				16#3: (* RAID sets state and info *)
					CASE MDP_Read.stMDP_DynAddr.nSubIdx	OF
					1:
						MEMCPY(ADR(SetState), ADR(DstBuf[0]), 1);
						MEMCPY(ADR(SetInfo), ADR(DstBuf[1]), 1);
						MDP_Read.stMDP_DynAddr.nSubIdx		:= 0;
						MDP_Read.stMDP_DynAddr.nTableId		:= 16#A;
					END_CASE


				16#A: (* Drives state  *)
					CASE MDP_Read.stMDP_DynAddr.nSubIdx	OF
					0:
						MEMCPY(ADR(CountDrives), ADR(DstBuf), SIZEOF(CountDrives));
						MDP_Read.stMDP_DynAddr.nSubIdx		:= 1;

					1..255:
						MEMCPY(ADR(DriveSTATE), ADR(DstBuf), 1);
						MDP_Read.stMDP_DynAddr.nSubIdx	:= MDP_Read.stMDP_DynAddr.nSubIdx + 1;
						IF MDP_Read.stMDP_DynAddr.nSubIdx > CountDrives
							OR MDP_Read.stMDP_DynAddr.nSubIdx > MAX_DRIVE
						THEN
							Busy							:= FALSE;
							Done							:= TRUE;
							state							:= 99;
						END_IF

					END_CASE

				ELSE
					Busy									:= FALSE;
					Done									:= TRUE;
					state									:= 99;
				END_CASE

				MDP_Read(
					stMDP_DynAddr	:= ,(* address to request subindex Count of AdressList *)
					pDstBuf			:= ADR(DstBuf),
					cbDstBufLen		:= SIZEOF(DstBuf),
					bExecute		:= NOT MDP_Read.bBusy AND state = 2,
					tTimeout		:= Timeout,
					sAmsNetId		:= AmsNetId,
					bBusy			=> ,
					bError			=> ,
					nErrId			=> );
			END_IF
		END_IF

	99: ;

	ELSE
		;
	END_CASE

	(* reset state for next start *)
	IF NOT Execute
		AND state = 99
	THEN
		state												:= 0;
	END_IF

(****************************************************************************************************)

END_FUNCTION_BLOCK

// POUs/IpcDiag/MDP/InfoModuls/MDP_ReadModulList
{attribute 'no_check'}
FUNCTION_BLOCK MDP_ReadModulList EXTENDS FbBase
VAR_INPUT
	AmsNetId												: 	T_AmsNetId := '';	//AmsNetId as text
	Timeout													:	TIME := DEFAULT_ADS_TIMEOUT;	//Ads timeout
END_VAR                     								
VAR_OUTPUT                  								
	ModulCount												:	USINT;	//number of modules
	ModulType												:	ARRAY[0..255] OF E_MDP_ModuleType; //Index = Modul ID
	ErrorGrp												:	E_MDP_ErrGroup := eMDP_Err_NoError;
END_VAR                     								
VAR                         								
	MDP_Read												: 	FB_MDP_Read		:= (stMDP_DynAddr := (nArea := INT_TO_BYTE(eMDP_Area_DeviceArea), nModuleId := 16#02, nTableId := 16#00, nFlag := 16#00, nSubIdx := 16#00));
	SplitErrorId											:	FB_MDP_SplitErrorID;
	dwData													:	ARRAY [1..2] OF WORD;
END_VAR

(* Read list ob available moduls			V1.0	*)
(****************************************************)

(* Start read ************************************************)
	IF Execute
		AND state = 0
	THEN
		IF FALSE
		THEN (* Modultypen Liste *)
			MDP_Read.stMDP_DynAddr.nModuleId				:= 16#01;
		ELSE (* Modul ID Liste *)               			
			MDP_Read.stMDP_DynAddr.nModuleId				:= 16#02;
		END_IF                                  			
		MDP_Read.stMDP_DynAddr.nSubIdx						:= 0;
		MEMSET(ADR(ModulType),0,SIZEOF(ModulType));
		ModulCount											:= 0;
		Busy												:= TRUE;
		Done												:= FALSE;
		Error												:= FALSE;
		ErrorId												:= 0;
		ErrorGrp											:= eMDP_Err_NoError;
		
		MDP_Read(
			stMDP_DynAddr	:= ,		(* address to request subindex Count of AdressList *)
			pDstBuf			:= ADR(dwData),
			cbDstBufLen		:= SIZEOF(dwData),
			bExecute		:= FALSE,
			tTimeout		:= Timeout,
			sAmsNetId		:= AmsNetId,
			bBusy			=> ,
			bError			=> ,
			nErrId			=> );

		MDP_Read(bExecute	:= TRUE);
		state												:= 1;
	ELSIF NOT Execute
		AND State = 99
	THEN
		state												:= 0;
		Busy												:= FALSE;
		Done												:= FALSE;
		Error												:= FALSE;
		ErrorId												:= 0;
		ErrorGrp											:= eMDP_Err_NoError;
	END_IF


	CASE state OF
	0:
		;
	1:
		MDP_Read(pDstBuf := ADR(dwData), cbDstBufLen := SIZEOF(dwData));
		IF NOT MDP_Read.bBusy
		THEN
			IF MDP_Read.bError AND MDP_Read.bExecute
			THEN
				Busy										:= FALSE;
				Error										:= TRUE;
				SplitErrorId(
					nErrID		:= MDP_Read.nErrID,
					eErrGroup	=> ErrorGrp ,
					nErrCode	=> ErrorId);
				state										:= 99;
				MDP_Read(bExecute := FALSE);
			ELSE
				IF ModulCount = 0
				THEN (* Init Modul count *)
					ModulCount								:= WORD_TO_USINT(dwData[1]);
				ELSIF MDP_Read.stMDP_DynAddr.nSubIdx > 0
				THEN (* copy emlement dat					a *)
					ModulType[MDP_Read.stMDP_DynAddr.nSubIdx - 1] :=  dwData[2];					
				END_IF
				MDP_Read(bExecute := FALSE);
				MDP_Read.stMDP_DynAddr.nSubIdx:= MDP_Read.stMDP_DynAddr.nSubIdx + 1;
				IF MDP_Read.stMDP_DynAddr.nSubIdx > ModulCount
					OR MDP_Read.stMDP_DynAddr.nSubIdx > 255
				THEN
					Busy									:= FALSE;
					Done									:= TRUE;
					state									:= 99;
				ELSE
					MDP_Read(bExecute := TRUE,	pDstBuf	:= ADR(dwData), cbDstBufLen := SIZEOF(dwData));
				END_IF
			END_IF

		END_IF

	99: ;

	ELSE
		;
	END_CASE

	(* reset state for next start *)
	IF NOT Execute
		AND state = 99
	THEN
		state												:= 0;
	END_IF

(****************************************************************************************************)

END_FUNCTION_BLOCK

// POUs/IpcDiag/MDP/InfoModuls/MDP_SiliconDrives
{attribute 'no_check'}
FUNCTION_BLOCK MDP_SiliconDrives  EXTENDS FbBase
VAR_OUTPUT CONSTANT
	MIN_DRIVES												:	INT := 1;
	MAX_DRIVES												:	INT := 4;
END_VAR                 									
VAR_INPUT               									
	AmsNetId												: 	T_AmsNetId := '';	//AmsNetId as text
	Timeout													:	TIME := DEFAULT_ADS_TIMEOUT;	//Ads timeout
END_VAR                 									
VAR_OUTPUT              									
	TotEraseCounts											:  ARRAY[MIN_DRIVES..MAX_DRIVES] OF	T_LARGE_INTEGER;	//total number erase operations
	Usage													:	ARRAY[MIN_DRIVES..MAX_DRIVES] OF	UINT;	//usage of drive in %
	NoOfSpares												:	ARRAY[MIN_DRIVES..MAX_DRIVES] OF	UINT;	//number of partitions
	SparedUsed												:	ARRAY[MIN_DRIVES..MAX_DRIVES] OF	UINT;	//usage of partitions
	Count													:	INT; 	//number of drives
	NoSiliconDrives											:	BOOL := FALSE;	//should be TRUE if there is no SSD drive in use
	ErrorGrp												:	E_MDP_ErrGroup := eMDP_Err_NoError;
END_VAR
VAR
	idx														:	INT := 1;
	MDP_ScanModules											:	FB_MDP_ScanModules := ( nModuleType 	:= eMDP_ModT_SiliconDrive , iModIdx		:= 0);
	MDP_Read												: 	FB_MDP_ReadModuleContent;
	SplitErrorId											:	FB_MDP_SplitErrorID;
	DstBuf													:	ARRAY[0..8] OF BYTE;
END_VAR

	(* Read CPU Information 					V1.0	*)
	(****************************************************)

(* Start Read *******************************************************)
	IF Execute
		AND state = 0
	THEN
		MEMSET(ADR(TotEraseCounts),0,SIZEOF(TotEraseCounts));
		MEMSET(ADR(Usage),0,SIZEOF(Usage));
		MEMSET(ADR(NoOfSpares),0,SIZEOF(NoOfSpares));
		MEMSET(ADR(SparedUsed),0,SIZEOF(SparedUsed));
	
		NoSiliconDrives										:= FALSE;
		Count												:= 0;
		Busy												:= TRUE;
		Done												:= FALSE;
		Error												:= FALSE;
		ErrorId												:= 0;
		ErrorGrp											:= eMDP_Err_NoError;
		MDP_Read(bExecute := FALSE);
		MDP_ScanModules(
			bExecute		:= NOT MDP_ScanModules.bExecute,
			nModuleType		:= eMDP_ModT_SiliconDrive,
			iModIdx			:= 0,
			tTimeout		:= timeout,
			sAmsNetId		:= AmsNetId,
			bBusy			=> ,
			bError			=> ,
			nErrID			=> ,
			nDynModuleId	=> ,
			iModuleTypeCount=> ,
			iModuleCount	=> );
		MDP_ScanModules(bExecute := TRUE);
		
		state												:= 1;
	ELSIF NOT Execute
		AND State = 99
	THEN
		state												:= 0;
		Busy												:= FALSE;
		Done												:= FALSE;
		Error												:= FALSE;
		ErrorId												:= 0;
		ErrorGrp											:= eMDP_Err_NoError;
	END_IF


	CASE state OF
	0:
		;
	1:
		MDP_ScanModules();
		IF NOT MDP_ScanModules.bBusy
		THEN
			IF MDP_ScanModules.bError
			THEN
				IF MDP_ScanModules.nErrID = 16#EC800002
				THEN
					Busy									:= FALSE;
					Done									:= TRUE;
					NoSiliconDrives							:= TRUE;
				ELSE

					Busy									:= FALSE;
					Error									:= TRUE;
					SplitErrorId(
						nErrID		:= MDP_ScanModules.nErrID,
						eErrGroup	=> ErrorGrp ,
						nErrCode	=> ErrorId);
				END_IF
				state										:= 99;
				MDP_ScanModules(bExecute := FALSE);
			ELSE
				Count										:= MDP_ScanModules.iModuleTypeCount;
				MDP_Read.stMDP_DynAddr.nArea				:= 16#8;
				MDP_Read.stMDP_DynAddr.nModuleId			:= MDP_ScanModules.nDynModuleId;
				MDP_Read.stMDP_DynAddr.nSubIdx				:= 0;
				MDP_Read.stMDP_DynAddr.nTableId				:= 1;
				MDP_Read(bExecute := FALSE);
				idx											:= 1;
				
				IF Count <= 0
				THEN
					Busy									:= FALSE;
					Done									:= TRUE;
					state									:= 99;
				ELSE
					state									:= 2;
				END_IF
			END_IF

		END_IF

	2:
		MDP_Read( pDstBuf:= ADR(DstBuf), cbDstBufLen:= SIZEOF(DstBuf));
		IF NOT MDP_Read.bBusy
		THEN
			IF MDP_Read.bError AND MDP_Read.bExecute
			THEN
				Busy										:= FALSE;
				Error										:= TRUE;
				SplitErrorId(
					nErrID		:= MDP_Read.nErrID,
					eErrGroup	=> ErrorGrp ,
					nErrCode	=> ErrorId);
				state										:= 99;
				MDP_Read(bExecute := FALSE);
			ELSE
				MDP_Read(bExecute := FALSE);
				CASE MDP_Read.stMDP_DynAddr.nSubIdx OF
				0:
					MDP_Read.stMDP_DynAddr.nSubIdx			:= 1;

				1:
					MEMCPY(ADR(TotEraseCounts[idx]), ADR(DstBuf), MIN(MDP_Read.nCount, SIZEOF(TotEraseCounts[MIN_DRIVES])));
					MDP_Read.stMDP_DynAddr.nSubIdx			:= 2;

				2:
					MEMCPY(ADR(Usage[idx]), ADR(DstBuf), SIZEOF(Usage[MIN_DRIVES]));
					MDP_Read.stMDP_DynAddr.nSubIdx			:= 3;

				3:
					MEMCPY(ADR(NoOfSpares[idx]), ADR(DstBuf), SIZEOF(NoOfSpares[MIN_DRIVES]));
					MDP_Read.stMDP_DynAddr.nSubIdx			:= 4;

				4:
					MEMCPY(ADR(SparedUsed[idx]), ADR(DstBuf), SIZEOF(SparedUsed[MIN_DRIVES]));
					MDP_Read.stMDP_DynAddr.nModuleId		:= MDP_Read.stMDP_DynAddr.nModuleId + 1;
					idx										:= idx + 1;
					MDP_Read.stMDP_DynAddr.nSubIdx			:= 1;
					IF idx > Count
						OR idx > MAX_DRIVES
					THEN
						Busy								:= FALSE;
						Done								:= TRUE;
						state								:= 99;
					END_IF
				END_CASE

				MDP_Read(
					stMDP_DynAddr	:= ,		(* address to request subindex Count of AdressList *)
					pDstBuf			:= ADR(DstBuf),
					cbDstBufLen		:= SIZEOF(DstBuf),
					bExecute		:= NOT MDP_Read.bBusy AND state = 2,
					tTimeout		:= Timeout,
					sAmsNetId		:= AmsNetId,
					bBusy			=> ,
					bError			=> ,
					nErrId			=> );

			END_IF
		END_IF

	99: ;

	ELSE
		;
	END_CASE

	(* reset state for next start *)
	IF NOT Execute
		AND state = 99
	THEN
		state												:= 0;
	END_IF

(****************************************************************************************************)

END_FUNCTION_BLOCK

// POUs/IpcDiag/MDP/InfoModuls/MDP_UPS
{attribute 'no_check'}
FUNCTION_BLOCK MDP_UPS EXTENDS FbBase
VAR_OUTPUT CONSTANT
(* Battery Power Status *)
	PS_UNKNOWN												:	INT := 0;
	PS_ONLINE												:	INT := 1;
	PS_ONBATTERIES											:	INT := 2;
	                    									
(* Com Status *)        									
	CS_UNKNOWN												:	INT := 0;
	CS_OK													:	INT := 1;
	CS_ERROR												:	INT := 2;

(* Battery Power Status *)
	BS_UNKNOWN												:	INT := 0;
	BS_OK													:	INT := 1;
	BS_CHANGE_BATTERY										:	INT := 2;
	
END_VAR
VAR_INPUT
	AmsNetId												: 	T_AmsNetId := '';	//AmsNetId
	Timeout													:	TIME := DEFAULT_ADS_TIMEOUT;	//Ads timeout
END_VAR
VAR_OUTPUT
(* UPS Data *)              								
	Model													:	STRING(30);	//model name
	VendorName												:	STRING(30);	//vendor name
	PowerStatus												:	INT := PS_UNKNOWN;
	ComStatus												:	INT := CS_UNKNOWN;
	BatteryStatus											:	INT := BS_UNKNOWN;
	BatteryCapacity											:	USINT; 		//in %
	BatteryRuntime											:	UDINT; 		//in sec
	PersPowerFailCounter									:	BOOL;		//TRUE when persistent power fail counter is activated
	PowerFailCounter										:	UDINT;		//number of power fails
	FanError												:	BOOL;		//Fan has error
	NoBattery												:	BOOL;		//No battery connected
	ErrorGrp												:	E_MDP_ErrGroup := eMDP_Err_NoError;

END_VAR                     								
VAR                         								
	idx														:	INT := 1;
	MDP_ScanModules											:	FB_MDP_ScanModules := ( nModuleType 	:= eMDP_ModT_UPS , iModIdx		:= 0);
	MDP_Read												: 	FB_MDP_Read;
	SplitErrorId											:	FB_MDP_SplitErrorID;
	DstBuf													:	ARRAY[0..31] OF BYTE;
END_VAR

	(* Read UPS Information 							V1.0	*)
	(***************************************************)

(* Start Read *******************************************************)
	IF Execute
		AND state = 0
	THEN
		Model												:= '';
		VendorName											:= '';
		PowerStatus											:= PS_UNKNOWN;
		ComStatus											:=	CS_UNKNOWN;
		BatteryStatus										:=	BS_UNKNOWN;
		BatteryCapacity										:= 0;
		BatteryRuntime										:= 0;
		PowerFailCounter									:= 0;
		PersPowerFailCounter								:= FALSE;
		FanError											:= FALSE;
		NoBattery											:= FALSE;
		Busy												:= TRUE;
		Done												:= FALSE;
		Error												:= FALSE;
		ErrorId												:= 0;
		ErrorGrp											:= eMDP_Err_NoError;
		MDP_Read(bExecute := FALSE);
		MDP_ScanModules(
			bExecute		:= NOT MDP_ScanModules.bExecute,
			nModuleType		:= eMDP_ModT_UPS,
			iModIdx			:= 0,
			tTimeout		:= timeout,
			sAmsNetId		:= AmsNetId,
			bBusy			=> ,
			bError			=> ,
			nErrID			=> ,
			nDynModuleId	=> ,
			iModuleTypeCount=> ,
			iModuleCount	=> );
			
		MDP_ScanModules(bExecute := TRUE);
		
		state												:= 1;
	ELSIF NOT Execute
		AND State = 99
	THEN
		state												:= 0;
		Busy												:= FALSE;
		Done												:= FALSE;
		Error												:= FALSE;
		ErrorId												:= 0;
		ErrorGrp											:= eMDP_Err_NoError;
	END_IF


	CASE state OF
	0:
		;
	1:
		MDP_ScanModules();
		IF NOT MDP_ScanModules.bBusy
		THEN
			IF MDP_ScanModules.bError
			THEN
				Busy										:= FALSE;
				Error										:= TRUE;
				SplitErrorId(
					nErrID		:= MDP_ScanModules.nErrID,
					eErrGroup	=> ErrorGrp ,
					nErrCode	=> ErrorId);
				state										:= 99;
				MDP_ScanModules(bExecute := FALSE);
			ELSE
				MDP_Read(bExecute := FALSE);
				MDP_Read.stMDP_DynAddr.nArea				:= 16#8;
				MDP_Read.stMDP_DynAddr.nModuleId			:= MDP_ScanModules.nDynModuleId;
				MDP_Read.stMDP_DynAddr.nTableId				:= 1;
				MDP_Read.stMDP_DynAddr.nSubIdx				:= 0;
				state										:= 2;
			END_IF

		END_IF

	2:
		MDP_Read( pDstBuf	:= ADR(DstBuf), cbDstBufLen := SIZEOF(DstBuf));
		IF NOT MDP_Read.bBusy
		THEN
			IF MDP_Read.bError AND MDP_Read.bExecute
			THEN
				Busy										:= FALSE;
				Error										:= TRUE;
				SplitErrorId(
					nErrID		:= MDP_Read.nErrID,
					eErrGroup	=> ErrorGrp ,
					nErrCode	=> ErrorId);
				state										:= 99;
				MDP_Read(bExecute := FALSE);
			ELSE
				MDP_Read(bExecute := FALSE);
				CASE MDP_Read.stMDP_DynAddr.nSubIdx	OF
				0:
					MDP_Read.stMDP_DynAddr.nSubIdx			:= 1;

				1:
					MEMCPY(ADR(Model), ADR(DstBuf), SIZEOF(Model) - 1);
					MDP_Read.stMDP_DynAddr.nSubIdx			:= 2;

				2:
					MEMCPY(ADR(VendorName), ADR(DstBuf), SIZEOF(VendorName) - 1);
					MDP_Read.stMDP_DynAddr.nSubIdx			:= 7;

				7:
					MEMCPY(ADR(PowerStatus), ADR(DstBuf), 1);
					MDP_Read.stMDP_DynAddr.nSubIdx			:= 8;

				8:
					MEMCPY(ADR(ComStatus), ADR(DstBuf), 1);
					MDP_Read.stMDP_DynAddr.nSubIdx			:= 9;

				9:
					MEMCPY(ADR(BatteryStatus), ADR(DstBuf), 1);
					MDP_Read.stMDP_DynAddr.nSubIdx			:= 10;

				10:
					MEMCPY(ADR(BatteryCapacity), ADR(DstBuf), SIZEOF(BatteryCapacity));
					MDP_Read.stMDP_DynAddr.nSubIdx			:= 11;

				11:
					MEMCPY(ADR(BatteryRuntime), ADR(DstBuf), SIZEOF(BatteryRuntime));
					MDP_Read.stMDP_DynAddr.nSubIdx			:= 12;

				12:
					MEMCPY(ADR(PersPowerFailCounter), ADR(DstBuf), SIZEOF(PersPowerFailCounter));
					MDP_Read.stMDP_DynAddr.nSubIdx			:= 13;

				13:
					MEMCPY(ADR(PowerFailCounter), ADR(DstBuf), SIZEOF(PowerFailCounter));
					MDP_Read.stMDP_DynAddr.nSubIdx			:= 14;

				14:
					MEMCPY(ADR(FanError), ADR(DstBuf), SIZEOF(FanError));
					MDP_Read.stMDP_DynAddr.nSubIdx			:= 15;

				15:
					MEMCPY(ADR(NoBattery), ADR(DstBuf), SIZEOF(NoBattery));
					Busy									:= FALSE;
					Done									:= TRUE;
					state									:= 99;
                                                        	
				ELSE                                    	
					Busy									:= FALSE;
					Done									:= TRUE;
					state									:= 99;
				END_CASE

				MDP_Read(
					stMDP_DynAddr	:= ,(* address to request subindex Count of AdressList *)
					pDstBuf			:= ADR(DstBuf),
					cbDstBufLen		:= SIZEOF(DstBuf),
					bExecute		:= NOT MDP_Read.bBusy AND state = 2,
					tTimeout		:= Timeout,
					sAmsNetId		:= AmsNetId,
					bBusy			=> ,
					bError			=> ,
					nErrId			=> );
			END_IF
		END_IF

	99: ;

	ELSE
		;
	END_CASE

	(* reset state for next start *)
	IF NOT Execute
		AND state = 99
	THEN
		state												:= 0;
	END_IF

(****************************************************************************************************)

END_FUNCTION_BLOCK

// POUs/IpcDiag/MDP/MDP_Info
{attribute 'no_check'}
//Wrapper for available MDP_xxxx FBs of the lib, based on Beckhoff MDP - invalid values are reported via EventLogger 
//based on Tc2_MDP.lib - please see Beckhoff documentation for further information about Tc2_MDP.lib (IPC diagnostics)
FUNCTION_BLOCK MDP_Info EXTENDS FbBase
VAR_OUTPUT CONSTANT
	FNC_READ_ALL											:	INT := 0;
	FNC_READ_MOD_LIST										:	INT := 1;
	FNC_READ_MB												:	INT := 2;
	FNC_READ_CPU											:	INT := 3;
	FNC_READ_FAN											:	INT := 4;
	FNC_READ_SD												:	INT := 5;
	FNC_READ_RAID											:	INT := 6;
	FNC_READ_UPS											:	INT := 7;
END_VAR                 									
VAR_INPUT               									
	AmsNetId												: 	T_AmsNetId := '';	//AmsNetId as text
	Timeout													:	TIME := DEFAULT_ADS_TIMEOUT; //Ads timeout
	Fnc														:	INT (FNC_READ_ALL..FNC_READ_UPS) := FNC_READ_ALL; //select function to be read
(* Components *)            								
	ModList													:	MDP_ReadModulList;	//see content in FB
	MB														:	MDP_Mainboard;		//see content in FB
	CPU														:	MDP_CPU;			//see content in FB
	FAN														:	MDP_Fan;			//see content in FB
	SD														:	MDP_SiliconDrives;	//see content in FB
	RAID													:	MDP_RaidSimple;		//see content in FB
	UPS														:	MDP_UPS;			//see content in FB
END_VAR                     								
VAR_OUTPUT                  								
	TotalCycleTime											:	TIME;	//Cylce time to execute function block with mode read all        
	ErrorGrp												:	E_MDP_ErrGroup;
	ErrorFnc												:	STRING(15);
END_VAR
VAR
	MemFnc													:	INT;
	MemExecute												:	BOOL;
	MemErrorFnc												:	STRING(15);
	MemErrorid												:	UDINT;
	MemErrorGrp												:	E_MDP_ErrGroup;
	MemTimeStartCycle										:	TIME;
END_VAR

	(* Execute all available MDP_xxxxx fb 			*)
	(************************************************)

(* Sequence ********************************************)
	IF Execute
		AND state = 0
	THEN
		ReadAll(Execute	:= Execute);
	ELSIF state <> 0
	THEN
		ReadAll(Execute	:= Execute);
	END_IF

(*****************************************************************************)

METHOD PUBLIC readAll : BOOL //Return value = TRUE if busy;
VAR_INPUT
	Execute													:	BOOL;
END_VAR
	THIS^.Execute											:= Execute;

	IF Execute
		AND State = 0
	THEN
		MemFnc												:= Fnc;
		CASE Fnc OF                                     	
		FNC_READ_MOD_LIST:		state						:= 10;
		FNC_READ_MB:			state						:= 20;
		FNC_READ_CPU:			state						:= 30;
		FNC_READ_FAN:			state						:= 40;
		FNC_READ_SD:			state						:= 50;
		FNC_READ_RAID:	 		state						:= 60;
		FNC_READ_UPS:	 		state						:= 70;
		ELSE (* Read All *)
			MemFnc											:= FNC_READ_ALL;
			state											:= 10;
		END_CASE
		MemTimeStartCycle									:= TIME();
		Busy												:= TRUE;
		Done												:= FALSE;
		Error												:= FALSE;
		Errorid												:= 0;
		ErrorFnc											:= '';
		ErrorGrp											:= eMDP_Err_NoError;
		MemExecute											:= FALSE;
		MemErrorid											:= 0;
		MemErrorFnc											:= '';
		MemErrorGrp											:= eMDP_Err_NoError;
	ELSIF NOT Execute
		AND State = 99
	THEN
		Busy												:= FALSE;
		Done												:= FALSE;
		Error												:= FALSE;
		Errorid												:= 0;
		ErrorFnc											:= '';
		ErrorGrp											:= eMDP_Err_NoError;
		MemExecute											:= FALSE;
		MemErrorid											:= 0;
		MemErrorFnc											:= '';
		MemErrorGrp											:= eMDP_Err_NoError;
		ReadModList(FALSE);     						
		ReadMB(FALSE);
		ReadCPU(FALSE);
		ReadFAN(FALSE);
		ReadSD(FALSE);
		ReadRaid(FALSE);
	END_IF

	CASE state OF
	10:

		MemExecute											:= TRUE;
		ReadModList(MemExecute);
		IF NOT ModList.Busy
		THEN
			IF MemFnc = FNC_READ_ALL
			THEN
				IF Error AND MemErrorid = 0 
				THEN
					MemErrorId								:= Errorid; 
					MemErrorFnc 							:= CONCAT('ReadModList Fnc:',TO_STRING(FNC_READ_MOD_LIST)); 
					MemErrorGrp 							:= ErrorGrp;
				END_IF              						
				Busy										:= TRUE;
				Done										:= FALSE;
				Error										:= FALSE;
				Errorid										:= 0;
				ErrorGrp									:= eMDP_Err_NoError;
				state										:= 20;
			ELSE                    						
				state										:= 99;
			END_IF
		END_IF

	20:
		MemExecute											:= TRUE;
		ReadMB(MemExecute);
		IF NOT MB.Busy
		THEN
			IF MemFnc = FNC_READ_ALL
			THEN
				IF Error AND MemErrorid = 0 
				THEN
					MemErrorId								:= Errorid; 
					MemErrorFnc 							:= CONCAT('ReadMB Fnc: ',TO_STRING(FNC_READ_MB));  
					MemErrorGrp 							:= ErrorGrp;
				END_IF              						
				Busy										:= TRUE;
				Done										:= FALSE;
				Error										:= FALSE;
				Errorid										:= 0;
				ErrorGrp									:= eMDP_Err_NoError;
				state										:= 30;
			ELSE                    						
				state										:= 99;
			END_IF                  	
		END_IF

	30:
		MemExecute											:= TRUE;
		ReadCPU(MemExecute);
		IF NOT CPU.Busy
		THEN
			IF MemFnc = FNC_READ_ALL
			THEN
				IF Error AND MemErrorid = 0 THEN
					MemErrorId								:= Errorid; 
					MemErrorFnc 							:= CONCAT('ReadCPU Fnc: ',TO_STRING(FNC_READ_CPU));  
					MemErrorGrp 							:= ErrorGrp;
				END_IF              						
				Busy										:= TRUE;
				Done										:= FALSE;
				Error										:= FALSE;
				Errorid										:= 0;
				ErrorGrp									:= eMDP_Err_NoError;
				state										:= 40;
			ELSE                    						
				state										:= 99;
			END_IF
		END_IF

	40:
		MemExecute											:= TRUE;
		ReadFan(MemExecute);
		IF NOT Fan.Busy
		THEN
			IF MemFnc = FNC_READ_ALL
			THEN
				IF Error AND MemErrorid = 0 
				THEN
					MemErrorId								:= Errorid; 
					MemErrorFnc 							:= CONCAT('ReadFan Fnc: ',TO_STRING(FNC_READ_FAN));  
					MemErrorGrp 							:= ErrorGrp;
				END_IF              						
				Busy										:= TRUE;
				Done										:= FALSE;
				Error										:= FALSE;
				Errorid										:= 0;
				ErrorGrp									:= eMDP_Err_NoError;
				state										:= 50;
			ELSE                    						
				state										:= 99;
			END_IF
		END_IF

	50:
		MemExecute											:= TRUE;		
		ReadSD(MemExecute);
		
		IF NOT SD.Busy
		THEN
			IF MemFnc = FNC_READ_ALL
			THEN
				IF Error AND MemErrorid = 0 
				THEN				
					MemErrorId								:= Errorid; 
					MemErrorFnc 							:= CONCAT('ReadSD Fnc: ',TO_STRING(FNC_READ_SD)); 
					MemErrorGrp 							:= ErrorGrp;
				END_IF              						
				Busy										:= TRUE;
				Done										:= FALSE;
				Error										:= FALSE;
				Errorid										:= 0;
				ErrorGrp									:= eMDP_Err_NoError;
				state										:= 60;
			ELSE                    						
				state										:= 99;
			END_IF                  	
		END_IF

	60:
		MemExecute											:= TRUE;
		ReadRaid(MemExecute);
		IF NOT Raid.Busy
		THEN
			IF MemFnc = FNC_READ_ALL
			THEN
				IF Error AND MemErrorid = 0 
				THEN
					MemErrorId								:= Errorid; 
					MemErrorFnc 							:= CONCAT('ReadRaid Fnc: ',TO_STRING(FNC_READ_RAID));
					MemErrorGrp 							:= ErrorGrp;
				END_IF              						
				Busy										:= TRUE;
				Done										:= FALSE;
				Error										:= FALSE;
				Errorid										:= 0;
				ErrorGrp									:= eMDP_Err_NoError;
				state										:= 70;
			ELSE                    						
				state										:= 99;
			END_IF
		END_IF

	70:
		MemExecute											:= TRUE;
		ReadUPS(MemExecute);
		IF NOT UPS.Busy
		THEN
			IF TRUE
			THEN
				IF Error AND MemErrorid = 0 
				THEN
					MemErrorId								:= Errorid; 
					MemErrorFnc 							:= CONCAT('ReadUPS Fnc: ',TO_STRING(FNC_READ_UPS));
					MemErrorGrp 							:= ErrorGrp;
				END_IF
				Busy										:= FALSE;
				Done										:= MemErrorId = 0;
				Error										:= MemErrorId <> 0;
				Errorid										:= MemErrorid;
				ErrorFnc									:= MemErrorFnc;
				ErrorGrp									:= MemErrorGrp;
				state										:= 99;
			ELSE                    						
				state										:= 99;
			END_IF
		END_IF

	99:;
	
	END_CASE

	IF state = 99
	THEN
		TotalCycleTime	 									:= TIME() - MemTimeStartCycle;
		IF NOT Execute
		THEN
			state											:= 0;
			ReadModList(FALSE);         					
			ReadMB(FALSE);              					
			ReadCPU(FALSE);             					
			ReadFAN(FALSE);             					
			ReadSD(FALSE);              					
			ReadRaid(FALSE);            					
			ReadUPS(FALSE);             	
		END_IF                          	
	END_IF                              	
	                                    	
	ReadAll													:= Busy;

(***********************************************************************************)
END_METHOD

METHOD PUBLIC readCPU : BOOL //Return value = TRUE if busy
VAR_INPUT
	Execute													:	BOOL;
END_VAR
THIS^.Execute												:= Execute;

CPU(
	Execute				:= MemExecute OR Execute,
	AmsNetId			:= AmsNetId,
	Timeout				:= Timeout,
	MIN_CPU				=> ,
	MAX_CPU				=> ,
	Busy				=> Busy,
	Done				=> Done,
	Error				=> Error,
	ErrorId				=> Errorid,
	ErrorGrp 			=> ErrorGrp,
	Frequency			=> ,
	Usage				=> ,
	Temperature			=> ,
	AverageFrequency	=> ,
	AverageUsage		=> ,
	AverageTemperature	=> ,
	Count				=> );

MemExecute 													:= FALSE;
	        												
ReadCPU														:= Busy;
END_METHOD

METHOD PUBLIC readFan : BOOL //Return value = TRUE if busy
VAR_INPUT
	Execute													:	BOOL;
END_VAR
THIS^.Execute												:= Execute;

FAN(
	Execute		:= MemExecute OR Execute,
	AmsNetId	:= AmsNetid,
	Timeout		:= Timeout,
	MIN_FAN		=> ,
	MAX_FAN		=> ,
	Busy		=> Busy,
	Done		=> Done,
	Error		=> Error,
	ErrorId		=> ErrorId,
	ErrorGrp 	=> ErrorGrp,
	Speed		=> ,
	Count		=> );

MemExecute 													:= FALSE;
           												
ReadFan														:= Busy;
END_METHOD

METHOD PUBLIC readMB : BOOL //Return value = TRUE if busy
VAR_INPUT
	Execute													:	BOOL;
END_VAR
THIS^.Execute												:= Execute;

MB(
	Execute			:= MemExecute OR Execute,
	AmsNetId		:= AmsNetId,
	Timeout			:= Timeout,
	MIN_VOLTAGE		=> ,
	MAX_VOLTAGE		=> ,
	Busy			=> Busy,
	Done			=> Done,
	Error			=> Error,
	ErrorId			=> ErrorId,
	ErrorGrp		=> Errorgrp,
	MB_Type			=> ,
	SerielNo		=> ,
	ProdDate		=> ,
	BootCount		=> ,
	OpTime			=> ,
	MinBoardTemp	=> ,
	MaxBoardTemp	=> ,
	MinInputVolt	=> ,
	MaxInputVolt	=> ,
	MB_Temp			=> ,
	VoltLocation	=> ,
	VoltageValue	=> ,
	VoltageNominal	=> ,
	VoltCount		=> );

MemExecute 													:= FALSE;
            												
ReadMB														:= Busy;
END_METHOD

METHOD PUBLIC readModList : BOOL //Return value = TRUE if busy
VAR_INPUT
	Execute													:	BOOL;
END_VAR
THIS^.Execute												:= Execute;

ModList(
	Execute		:= MemExecute OR Execute,
	AmsNetId	:= AmsNetId,
	Timeout		:= Timeout,
	Busy		=> Busy,
	Done		=> done,
	Error		=> Error,
	ErrorId		=> ErrorId,
	ErrorGrp 	=> ErrorGrp );

MemExecute 													:= FALSE;
            												
ReadModList													:= Busy;
END_METHOD

METHOD PUBLIC readRaid : BOOL //Return value = TRUE if busy
VAR_INPUT
	Execute													: BOOL;
END_VAR
THIS^.Execute												:= Execute;

RAID(
	Execute			:= Execute OR MemExecute,
	AmsNetId		:= AmsNetId,
	Timeout			:= timeout,
	MIN_DRIVE		=> ,
	MAX_DRIVE		=> ,
	Busy			=> Busy,
	Done			=> done,
	Error			=> Error,
	ErrorId			=> ErrorId,
	ErrorGrp 		=> ErrorGrp,
	CntrState		=> ,
	CntrOfflReason	=> ,
	SetType			=> ,
	SetState		=> ,
	SetInfo			=> ,
	CountDrives		=> ,
	DriveSTATE		=> ,
	CountRAIDSets	=> );

MemExecute 													:= FALSE;
                											
ReadRaid													:= Busy;
END_METHOD

METHOD PUBLIC readSD : BOOL //Return value = TRUE if busy
VAR_INPUT
	Execute		:	BOOL;
END_VAR
THIS^.Execute												:= Execute;

SD(
	Execute			:= MemExecute OR Execute,
	AmsNetId		:= AmsNetid,
	Timeout			:= timeout,
	MIN_DRIVES		=> ,
	MAX_DRIVES		=> ,
	Busy			=> Busy,
	Done			=> Done,
	Error			=> Error,
	ErrorId			=> Errorid,
	ErrorGrp 		=> ErrorGrp,
	TotEraseCounts	=> ,
	Usage			=> ,
	NoOfSpares		=> ,
	SparedUsed		=> ,
	Count			=> );

MemExecute	 												:= FALSE;
                											
ReadSD														:= Busy;
END_METHOD

METHOD PUBLIC readUPS : Bool //Return value = TRUE if busy
VAR_INPUT
	Execute		:	BOOL;
END_VAR
THIS^.Execute												:= Execute;

UPS(
	Execute					:= MemExecute OR Execute,
	AmsNetId				:= AmsNetid,
	Timeout					:= timeout,
	Busy					=> Busy,
	Done					=> Done,
	Error					=> Error,
	ErrorId					=> Errorid,
	ErrorGrp				=> ErrorGrp,
	Model					=> ,
	VendorName				=> ,
	PowerStatus				=> ,
	ComStatus				=> ,
	BatteryStatus			=> ,
	BatteryCapacity			=> ,
	BatteryRuntime			=> ,
	PersPowerFailCounter	=> ,
	PowerFailCounter		=> ,
	FanError				=> ,
	NoBattery				=> );

MemExecute 													:= FALSE;
ReadUPS														:= Busy;
END_METHOD

END_FUNCTION_BLOCK

// POUs/IpcDiag/MDP/MDP_IpcDiag
{attribute 'no_check'}
//General IPC diagnosis based on Beckhoff MDP - invalid values are reported via EventLogger 
//based on Tc2_MDP.lib - please see Beckhoff documentation for further information about Tc2_MDP.lib (IPC diagnostics)
//EventHandlingGrp10 instance used inside
//Info:
// 0x   	a    	nn   	x   
// 0x   	8   	03   	1   
// a 	= Area Code (e.g. 8 = Configuration Area) 
// nn 	= Modul-ID (e.g. dynamic modul id from list F020) 
// x	= Tabel id (e.g. 1 = Table 0x8nn1 - NIC Properties at area code 8) 
FUNCTION_BLOCK MDP_IpcDiag
VAR CONSTANT
	MIN_CPU													:	INT := 1;
	MAX_CPU													:	INT := 4;
	                    									
	MIN_FAN													:	INT := 1;
	MAX_FAN													:	INT := 4;
	                    									
	MIN_VOLTAGE												:	INT := 1;
	MAX_VOLTAGE												:	INT := 8;		
END_VAR                 									
VAR_INPUT               									
	Enable													:	BOOL := FALSE;	//FB will be processed as long as enable is TRUE 
	CycleTime												:	TIME := T#100MS; //Delay between ads call to read a single value 
	AmsNetId												: 	T_AmsNetId := ''; //Ams net Id
	Timeout													: 	TIME := DEFAULT_ADS_TIMEOUT; //Ads timeout
{attribute 'displaymode':='bin'}
	FanMask													:	BYTE := 2#0000_0011; //Installed fans inside the PC 
	
//Threshold values 	    									
	MinSpeedFan												:	INT := 2500; 	//rpm
	MaxTempMB												:	INT := 85; 		//°C
	MaxTempCPU												:	INT := 100; 	//°C
	TempWarningThreshold									:	INT := 10; 		//°C
	VoltageFactor											:	LREAL := 0.7; 	//% of nominal voltage before an error occurs
END_VAR                 									
VAR_OUTPUT              										                									
	MB_Temp													:	INT; //Motherboard temp with one decimal digit  
	Voltage_Count											:	INT := 0; //count of voltage measurement points with one decimal digit 
	MB_NominalVoltage										:	ARRAY[MIN_VOLTAGE..MAX_VOLTAGE] OF INT; //in mV
	MB_Voltage												:	ARRAY[MIN_VOLTAGE..MAX_VOLTAGE] OF INT;  //in mV
	CPU_Count												:	INT := 0; //Readed number of CPUs
	CPU_Temp												:	ARRAY[MIN_CPU..MAX_CPU] OF INT; //cpu temperatur with one decimal digit
	FAN_Count												:	INT := 0; //Number of FANs in config. Note, the number may be two where only the second fan is p
	FAN_Speed												:	ARRAY[MIN_FAN..MAX_FAN] OF INT; //in rpm for each available fan
	OsImage													:	STRING; //Image version 
	ExecutionTime											:	TIME; 	//Cylce time to execute function block        
	Busy													:	BOOL;	//Busy is TRUE at the rising edge of Enable and stays TRUE as long as the FB is performing any action. 
	Valid													:	BOOL;	//data valid
	Error													:	BOOL;	//Rising edge of Error informs that an error occurred during the execution of the Function Block 
{attribute 'displaymode':='hex'}
	ErrorId													:	UDINT;	//Error identification - see documentation about IPC diagnostic for further detailed informantion 
	ErrorGrp												:	E_MDP_ErrGroup := eMDP_Err_NoError; //MDP Error code - see Beckhoff documentation MDP for further informantion
END_VAR	
VAR
(* cache variables ************************************************************)
	state													:	INT := 0;
	
	dwData													:	ARRAY [1..2] OF WORD;
	                    									
	MemLen													:	BYTE := 0;
	MemModIdMB												:	BYTE;
	MemModIdCPU												:	ARRAY[MIN_CPU..MAX_CPU] OF BYTE;
	MemModIdFan												:	ARRAY[MIN_FAN..MAX_FAN] OF BYTE;
	MEmModIdUPS												:	BYTE;
	MemMBSubIdxVoltage										:	ARRAY[MIN_VOLTAGE..MAX_VOLTAGE] OF BYTE;
	MemTimeStartCycle										:	TIME;
	MemErrState												:	INT := 0;
	
(* timer ***************************************************************************)
	TON_Cycle												:	TON;
	
(* function-blocks *****************************************************************)
	MDP_Read												: 	FB_MDP_Read		:= (tTimeout := DEFAULT_ADS_TIMEOUT, stMDP_DynAddr := (nArea := INT_TO_BYTE(eMDP_Area_DeviceArea), nModuleId := 16#02, nTableId := 16#00, nFlag := 16#00, nSubIdx := 16#00));
	SplitErrorId											:	FB_MDP_SplitErrorID;
	
(* internal used variables **********************************************************)
	i,k														:	INT;

END_VAR

(* MDP IPC diag compact						V1.1	*)
(****************************************************)

(* Sequence *******************************************************)
IF Enable
THEN
	CASE state OF
	0:	
		IF NOT MDP_Read.bBusy
			AND NOT Error
		THEN
			Busy											:= TRUE;
			Valid											:= FALSE;
		
			Fan_Count										:= 0;
			CPU_Count										:= 0;
			Voltage_Count									:= 0;
			MemLen											:= 0;
			MB_Temp											:= 0;
			MEMSET(ADR(MB_Voltage),0,SIZEOF(MB_Voltage));
			MEMSET(ADR(CPU_Temp),0,SIZEOF(CPU_Temp));
			MEMSET(ADR(FAN_Speed),0,SIZEOF(FAN_Speed));
			MEMSET(ADR(MemModIdCPU),0,SIZEOF(MemModIdCPU));
			MEMSET(ADR(MemModIdFan),0,SIZEOF(MemModIdFan));
			MEMSET(ADR(MemMBSubIdxVoltage),0,SIZEOF(MemMBSubIdxVoltage));
			MEMSET(ADR(MB_NominalVoltage),0,SIZEOF(MB_NominalVoltage));
			
			MDP_Read.stMDP_DynAddr.nArea					:= INT_TO_BYTE(eMDP_Area_GeneralArea);
			MDP_Read.stMDP_DynAddr.nModuleId				:= 16#00;
			MDP_Read.stMDP_DynAddr.nTableId					:= 16#0A;
			MDP_Read.stMDP_DynAddr.nSubIdx					:= 16#00;
                                                    			                                        		
			state											:= 1;
		ELSE
			MDP_Read(bExecute := FALSE);	
		END_IF
		
	1:
	//Read OS version 	
		MDP_Read(bExecute := TRUE , pDstBuf := ADR(OsImage), cbDstBufLen := SIZEOF(OsImage));
		IF NOT MDP_Read.bBusy
		THEN
			IF MDP_Read.bError AND MDP_Read.bExecute
			THEN
				Busy										:= FALSE;
				Error										:= TRUE;
				SplitErrorId(
					nErrID		:= MDP_Read.nErrID,
					eErrGroup	=> ErrorGrp ,
					nErrCode	=> ErrorId);
				MemErrState									:= state;		
				state										:= 99;
				MDP_Read(bExecute := FALSE);
			ELSE //Os Image readed
				k											:= UDINT_TO_INT(MDP_Read.nCount + 1);	
				OsImage[k]									:= 0; //Terminate string
				MDP_Read(bExecute := FALSE);	
				
				//Deveice area F + Modul Id 02 + Tabel Id = 0 -> Index 0xF020 – Modul ID Liste in deveice area
				MDP_Read.stMDP_DynAddr.nArea				:= INT_TO_BYTE(eMDP_Area_DeviceArea); //Index F
				MDP_Read.stMDP_DynAddr.nModuleId			:= 16#02; //Modul id 02 in Config area dynamic modul ids are used!
				MDP_Read.stMDP_DynAddr.nTableId				:= 16#00; //Table Id 0
				MDP_Read.stMDP_DynAddr.nSubIdx				:= 16#00; //Len = number of dyn moduls			
				state										:= 2;								
			END_IF
		END_IF		
		
	2: // search list with dynamic moduls
		MDP_Read(bExecute := TRUE, pDstBuf := ADR(dwData), cbDstBufLen := SIZEOF(dwData));
		IF NOT MDP_Read.bBusy
		THEN
			IF MDP_Read.bError AND MDP_Read.bExecute
			THEN
				Busy										:= FALSE;
				Error										:= TRUE;
				SplitErrorId(
					nErrID		:= MDP_Read.nErrID,
					eErrGroup	=> ErrorGrp ,
					nErrCode	=> ErrorId);
				MemErrState									:= state;	
				state										:= 99;
				MDP_Read(bExecute := FALSE);
			ELSE
				IF MemLen = 0
				THEN (* Init Modul count *)
					MemLen									:= WORD_TO_BYTE(dwData[1]);
				ELSIF MDP_Read.stMDP_DynAddr.nSubIdx > 0
				THEN (* copy emlement dat					a *)
					CASE dwData[2] OF //High word = Modul type, Low word = Modul Id
					Tc2_MDP.E_MDP_ModuleType.eMDP_ModT_Mainboard:
						MemModIdMB		 					:= WORD_TO_BYTE(dwData[1]);		

					Tc2_MDP.E_MDP_ModuleType.eMDP_ModT_UPS:
						MEmModIdUPS							:= WORD_TO_BYTE(dwData[1]);

					Tc2_MDP.E_MDP_ModuleType.eMDP_ModT_CPU:
						CPU_Count							:= CPU_Count + 1;
						MemModIdCPU[CPU_Count]				:= WORD_TO_BYTE(dwData[1]);

					Tc2_MDP.E_MDP_ModuleType.eMDP_ModT_Fan:
						Fan_Count							:= Fan_Count + 1;
						MemModIdFan[Fan_Count]				:= WORD_TO_BYTE(dwData[1]);
												
					ELSE
						; 
					END_CASE				
				END_IF
				MDP_Read(bExecute := FALSE);
				MDP_Read.stMDP_DynAddr.nSubIdx:= MDP_Read.stMDP_DynAddr.nSubIdx + 1;
				IF MDP_Read.stMDP_DynAddr.nSubIdx > MemLen
					OR MDP_Read.stMDP_DynAddr.nSubIdx > 255
				THEN
					state									:= SEL(MemModIdMB > 0 , 9 , 3);								
				ELSE
					MDP_Read(bExecute := TRUE,	pDstBuf	:= ADR(dwData), cbDstBufLen := SIZEOF(dwData));
				END_IF
			END_IF

		END_IF
				
	3: //reading motherboardconfig (SubIndex Voltage)
		MDP_Read.stMDP_DynAddr.nArea						:= INT_TO_BYTE(eMDP_Area_ConfigArea);
		MDP_Read.stMDP_DynAddr.nModuleId					:= INT_TO_BYTE(MemModIdMB);
		MDP_Read.stMDP_DynAddr.nTableId						:= 16#04;
		MDP_Read.stMDP_DynAddr.nSubIdx						:= 16#00;
		MemLen												:= 0;
		i													:= 0;
		
		MDP_Read(
			stMDP_DynAddr	:= ,		(* address to request subindex Count of AdressList *)
			pDstBuf			:= ADR(dwData[1]),
			cbDstBufLen		:= SIZEOF(dwData[1]),
			bExecute		:= NOT MDP_Read.bBusy,
			tTimeout		:= ,
			sAmsNetId		:= AmsNetId,
			bBusy			=> ,
			bError			=> ,
			nErrId			=> );	
			
		state												:= 4;	
	
	4: 
		MDP_Read(pDstBuf := ADR(dwData[1]), cbDstBufLen := SIZEOF(dwData[1]));
		IF NOT MDP_Read.bBusy
		THEN
			IF MDP_Read.bError AND MDP_Read.bExecute
			THEN
				Busy										:= FALSE;
				Error										:= TRUE;
				SplitErrorId(
					nErrID		:= MDP_Read.nErrID,
					eErrGroup	=> ErrorGrp ,
					nErrCode	=> ErrorId);
				MemErrState									:= state;		
				state										:= 99;
				MDP_Read(bExecute := FALSE);
			ELSE
				IF MemLen = 0
				THEN (* Init Entry count *)
					MemLen									:= WORD_TO_BYTE(dwData[1]);
				ELSE 
					MDP_Read(bExecute := FALSE);
					(* copy emlement data
						00 = LOCATION_UNKNOWN
						01 = LOCATION_OTHER
						02 = LOCATION_PROCESSOR
						03 = LOCATION_DISK
						04 = LOCATION_SYSTEM_MANAGEMENT_MODULE
						05 = LOCATION_MOTHERBOARD
						06 = LOCATION_MEMORY_MODULE
						07 = LOCATION_POWER_SUPPLY
						08 = LOCATION_ADDIN_CARD
						09 = LOCATION_FRONT_PANEL_BOARD
						10 = LOCATION_BACK_PANEL_BOARD
						11 = LOCATION_PERIPHERIE
						12 = LOCATION_CHASSIS
						13 = LOCATION_BATTERY
						14 = LOCATION_UPS
						15 = LOCATION_GRAFFIC_BOARD
						16 = LOCATION_SUPERIO
						17 = LOCATION_CHIPSET
					*)

				
					CASE dwData[1] OF
					7, //PowerSupply			
					13: //Battery
						Voltage_Count						:= Voltage_Count + 1;
						MemMBSubIdxVoltage[Voltage_Count]	:= MDP_Read.stMDP_DynAddr.nSubIdx; 
					ELSE
						; 
					END_CASE			
					MDP_Read.stMDP_DynAddr.nSubIdx			:= MDP_Read.stMDP_DynAddr.nSubIdx + 1; 				
							
					IF MDP_Read.stMDP_DynAddr.nSubIdx > MemLen
						OR MDP_Read.stMDP_DynAddr.nSubIdx > 255
						OR Voltage_Count >= MAX_Voltage
					THEN
						IF Voltage_Count > 0
						THEN
							i 								:= MIN_VOLTAGE;
							MDP_Read.stMDP_DynAddr.nTableId	:= 16#06;
							MDP_Read.stMDP_DynAddr.nSubIdx	:= MemMBSubIdxVoltage[i];
							MDP_Read(bExecute := TRUE,	pDstBuf	:= ADR(dwData[1]), cbDstBufLen := SIZEOF(dwData[1]));												
							state							:= 5;				
						ELSE
							state							:= 9;	
						END_IF
				
					ELSE
						MDP_Read(bExecute := TRUE,	pDstBuf	:= ADR(dwData[1]), cbDstBufLen := SIZEOF(dwData[1]));
					END_IF
				END_IF
			END_IF

		END_IF	

	5:	//Nominal Voltage lesen
		MDP_Read(pDstBuf := ADR(dwData[1]), cbDstBufLen := SIZEOF(dwData[1]));
		IF NOT MDP_Read.bBusy
		THEN
			IF MDP_Read.bError AND MDP_Read.bExecute
			THEN
				Busy										:= FALSE;
				Error										:= TRUE;
				SplitErrorId(
					nErrID		:= MDP_Read.nErrID,
					eErrGroup	=> ErrorGrp ,
					nErrCode	=> ErrorId);
				MemErrState									:= state;		
				state										:= 99;
				MDP_Read(bExecute := FALSE);
			ELSE //Nominal Volage
				MDP_Read(bExecute := FALSE);
				MB_NominalVoltage[i]						:= WORD_TO_INT(dwData[1]); 
				i 											:= i + 1;
				IF i > MAX_VOLTAGE
					OR i > Voltage_Count
				THEN //Ende der Bearbeitung
					state									:= 9;								
				ELSE
					MDP_Read.stMDP_DynAddr.nSubIdx			:= MemMBSubIdxVoltage[i];
					MDP_Read(bExecute := TRUE,	pDstBuf	:= ADR(dwData[1]), cbDstBufLen := SIZEOF(dwData[1]));
				END_IF
			END_IF

		END_IF	
							
	//Start Cylce Read
	9: 	
		TON_Cycle(IN := FALSE);
		MemTimeStartCycle									:= T#0MS;
		i													:= 0;
		state												:= 10;	
		
	//Start lesen der Zyklischen Daten 
	10..90: 
		MDP_Read(pDstBuf := ADR(dwData[1]), cbDstBufLen := SIZEOF(dwData[1]));
		IF NOT MDP_Read.bBusy
		THEN			
			IF MDP_Read.bError AND MDP_Read.bExecute
			THEN
				Busy										:= FALSE;
				Error										:= TRUE;
				SplitErrorId(
					nErrID		:= MDP_Read.nErrID,
					eErrGroup	=> ErrorGrp ,
					nErrCode	=> ErrorId);
				MemErrState									:= state;	
				state										:= 99;
				MDP_Read(bExecute := FALSE);
			ELSIF NOT TON_Cycle.IN
			THEN		
				MDP_Read(bExecute := FALSE);
				CASE state OF
				10:
					MDP_Read.stMDP_DynAddr.nModuleId		:= MemModIdMB;
					MDP_Read.stMDP_DynAddr.nTableId			:= 16#01;
					MDP_Read.stMDP_DynAddr.nSubIdx			:= 10;
					dwData[1]								:= 0;	
					TON_Cycle.IN							:= MDP_Read.stMDP_DynAddr.nModuleId > 0;			
					state									:= 11;
								
				11: 
					MB_Temp									:= WORD_TO_INT(dwData[1]); //Daten sichern
					
					i 										:= MIN_VOLTAGE;	
					IF Voltage_Count > 0
					THEN					
						MDP_Read.stMDP_DynAddr.nModuleId	:= MemModIdMB;
						MDP_Read.stMDP_DynAddr.nTableId		:= 16#05;
						MDP_Read.stMDP_DynAddr.nSubIdx		:= MemMBSubIdxVoltage[i];
						TON_Cycle.IN						:= MDP_Read.stMDP_DynAddr.nModuleId > 0;	
					ELSE
						dwData[1]							:= 0;	
					END_IF						
					
					state									:= 12;		
			
				12:
					MB_Voltage[i]							:= WORD_TO_INT(dwData[1]); //Daten sichern
				
					i 										:= i + 1;	
					IF i > Voltage_Count
					THEN //CPUTemp lesen 
						i									:= MIN_CPU;
						MDP_Read.stMDP_DynAddr.nModuleId	:= MemModIdCPU[i];
						MDP_Read.stMDP_DynAddr.nTableId		:= 16#01;
						MDP_Read.stMDP_DynAddr.nSubIdx		:= 3;
						TON_Cycle.IN						:= MDP_Read.stMDP_DynAddr.nModuleId > 0;		
						state								:= 13;					
					ELSE //weiter Voltage lesen
						MDP_Read.stMDP_DynAddr.nModuleId	:= MemModIdMB;
						MDP_Read.stMDP_DynAddr.nTableId		:= 16#05;
						MDP_Read.stMDP_DynAddr.nSubIdx		:= MemMBSubIdxVoltage[i];	
						TON_Cycle.IN						:= MDP_Read.stMDP_DynAddr.nModuleId > 0;		
					END_IF								
			
				13: 
					CPU_Temp[i]								:= WORD_TO_INT(dwData[1]);
					
					i 										:= i + 1;	
					IF i > CPU_Count //Start next read
					THEN //Fan auslesen 	
						IF Fan_Count > 0
						THEN
							i								:= MIN_FAN;
							
							MDP_Read.stMDP_DynAddr.nModuleId:= MemModIdFan[i];
							MDP_Read.stMDP_DynAddr.nTableId	:= 16#01;
							MDP_Read.stMDP_DynAddr.nSubIdx	:= 1;		
							TON_Cycle.IN					:= MDP_Read.stMDP_DynAddr.nModuleId > 0;			
						ELSE
							dwData[1]						:= 0;				
						END_IF
						
						state								:= 14;
						
					ELSE //CPU weiter auslesen
						MDP_Read.stMDP_DynAddr.nModuleId	:= MemModIdCPU[i];
						MDP_Read.stMDP_DynAddr.nTableId		:= 16#01;
						MDP_Read.stMDP_DynAddr.nSubIdx		:= 3;		
						TON_Cycle.IN						:= MDP_Read.stMDP_DynAddr.nModuleId > 0;						
					END_IF			
				
				14: 
					FAN_Speed[i]							:= WORD_TO_INT(dwData[1]);
					
					i 										:= i + 1;	
					IF i > Fan_Count
					THEN //CPU Usage auslesen
						(*
						i									:= MIN_CPU;
						MDP_Read.stMDP_DynAddr.nModuleId	:= MemModIdCPU[i];
						MDP_Read.stMDP_DynAddr.nTableId		:= 16#01;
						MDP_Read.stMDP_DynAddr.nSubIdx		:= 2;
						*)
						TON_Cycle.IN						:= MDP_Read.stMDP_DynAddr.nModuleId > 0;		
					//	state								:= 15;
						state								:= 90;	//final state in this section		
					
					ELSE //Fan weiter auslesen
						MDP_Read.stMDP_DynAddr.nModuleId	:= MemModIdFan[i];
						MDP_Read.stMDP_DynAddr.nTableId		:= 16#01;
						MDP_Read.stMDP_DynAddr.nSubIdx		:= 1;
						TON_Cycle.IN						:= MDP_Read.stMDP_DynAddr.nModuleId > 0;						
					END_IF				
				
				(*
				15:
					CPU_Usage[i]							:= WORD_TO_USINT(dwData[1]);
					
					i 										:= i + 1;	
					IF i > CPUCount
					THEN //Ups status auslesen 	
						IF MEmModIdUPS <> 0
						THEN
							MDP_Read.stMDP_DynAddr.nModuleId:= MEmModIdUPS;
							MDP_Read.stMDP_DynAddr.nTableId	:= 16#01;
							MDP_Read.stMDP_DynAddr.nSubIdx	:= 7;	
							TON_Cycle.IN					:= MDP_Read.stMDP_DynAddr.nModuleId > 0;
						ELSE
							dwData[1]						:= 0;								
						END_IF					
						state								:= 16;	
						
					ELSE //CPU weiter auslesen
						MDP_Read.stMDP_DynAddr.nModuleId	:= MemModIdCPU[i];
						MDP_Read.stMDP_DynAddr.nTableId		:= 16#01;
						MDP_Read.stMDP_DynAddr.nSubIdx		:= 2;		
						TON_Cycle.IN						:= MDP_Read.stMDP_DynAddr.nModuleId > 0;						
					END_IF	
			
				16:
					UPS_PowerStatus							:= WORD_TO_INT(dwData[1]);
					state									:= state * -1;	
				*)
				ELSE //90			
					Valid									:= TRUE;
					ExecutionTime	 						:= TIME() - MemTimeStartCycle;
					MemTimeStartCycle 						:= T#0MS;
					state									:= 10;	
				END_CASE
			END_IF
			TON_Cycle(PT := CycleTime);
			MDP_Read(bExecute := TON_Cycle.Q,	pDstBuf	:= ADR(dwData), cbDstBufLen := SIZEOF(dwData));
			
			IF MDP_Read.bExecute 
			THEN 
				TON_Cycle(IN := FALSE); 		
			END_IF 
			
			IF MemTimeStartCycle = T#0MS
			THEN
				MemTimeStartCycle 							:= TIME();	
			END_IF
			
		END_IF
			
	//Error State	
	99:	
		; //Wait for disable
				
	ELSE
		;
	END_CASE
ELSE //Not Enable
	state													:= 0;
	Error													:= FALSE;
	ErrorId													:= 0;
	ErrorGrp												:= eMDP_Err_NoError;
	Busy													:= FALSE;
	Valid													:= FALSE;
	MDP_Read(bExecute := FALSE);

END_IF			

(****************************************************************************************************)

END_FUNCTION_BLOCK

// POUs/IpcDiag/MDP/MDP_IpcDiag_wEvents
{attribute 'no_check'}
//General IPC diagnosis based on Beckhoff MDP - invalid values are reported via EventLogger 
//based on Tc2_MDP.lib - please see Beckhoff documentation for further information about Tc2_MDP.lib (IPC diagnostics)
//EventHandlingGrp10 instance used inside
//Info:
// 0x   	a    	nn   	x   
// 0x   	8   	03   	1   
// a 	= Area Code (e.g. 8 = Configuration Area) 
// nn 	= Modul-ID (e.g. dynamic modul id from list F020) 
// x	= Tabel id (e.g. 1 = Table 0x8nn1 - NIC Properties at area code 8) 
FUNCTION_BLOCK MDP_IpcDiag_wEvents EXTENDS MDP_IpcDiag         									
VAR_INPUT               									
	ConfirmTrig												:	BOOL := FALSE;	//Resets error with rising edge
	SourceId												:	UDINT := 100001; //EventLogger source id - Initinal value collaborates with SOURCE_ID structure 

END_VAR                 									
VAR_OUTPUT              							
	EventStatus												:	DWORD;	//state of event
END_VAR	
VAR
(* function-blocks *****************************************************************)
	Event													:	EventHandlingGrp10:= (  
																	No := [(Class := TC2_SYSTEM.TCEVENTCLASS_ALARM),
																			(Class := TC2_SYSTEM.TCEVENTCLASS_ALARM),
																			(Class := TC2_SYSTEM.TCEVENTCLASS_ALARM),
																			(Class := TC2_SYSTEM.TCEVENTCLASS_ALARM),
																			(Class := TC2_SYSTEM.TCEVENTCLASS_ALARM),
																			(Class := TC2_SYSTEM.TCEVENTCLASS_ALARM),
																			(Class := TC2_SYSTEM.TCEVENTCLASS_ALARM),
																			(Class := TC2_SYSTEM.TCEVENTCLASS_ALARM),
																			(Class := TC2_SYSTEM.TCEVENTCLASS_WARNING),
																			(Class := TC2_SYSTEM.TCEVENTCLASS_WARNING)]);
	
(* internal used variables **********************************************************)

END_VAR

(* MDP IPC diag compact						V1.1	*)
(****************************************************)

(* call base *******************************************************)
	SUPER^();

	//Leave error state by confirm trigger too
	IF State = 99 AND ConfirmTrig
	THEN
		state											:= 0;
		Error											:= FALSE;
		ErrorId											:= 0;
		ErrorGrp										:= eMDP_Err_NoError;
		Busy											:= FALSE;
		Valid											:= FALSE;
		MDP_Read(bExecute := FALSE);						
	END_IF
	
(* Meldungen *******************************************************)
	_callEvents();

(******************************************************************)

METHOD _callEvents : BOOL
VAR_INPUT
END_VAR
	IF state = 90 
		OR ConfirmTrig AND Valid
	THEN //Nur nach lesen Ende auswerten
		event.no[1].Flag 									:= FALSE ; 
		event.no[2].Flag 									:= MAX(CPU_Temp[1],CPU_Temp[2]) > MaxTempCPU; event.no[2].Text1 := INT_TO_STRING(MAX(CPU_Temp[1],CPU_Temp[2])); 
		event.no[3].Flag 									:= MB_Temp > MaxTempMB; event.no[3].Text1 := INT_TO_STRING(MB_Temp); 
	
		IF Fan_Count > 0
		THEN
			event.no[4].Flag := FALSE;
			FOR k := MIN_FAN TO MIN(Fan_Count,MAX_FAN)
			DO
				IF FAN_Speed[k] < MinSpeedFan 
					AND_THEN GETBIT32(TO_DWORD(FanMask), TO_SINT(k-1)) //Only check for active marked fans
				THEN
					event.no[4].Text1 						:= INT_TO_STRING(k); 
					event.no[4].Text2 						:= INT_TO_STRING(FAN_Speed[k]); 				
					event.no[4].Flag 						:= TRUE;
					EXIT;
				END_IF
			END_FOR		 
		ELSE
			event.no[4].Flag 								:= FALSE;
		END_IF
		
		IF Voltage_Count > 0
		THEN
			event.no[5].Flag 								:= FALSE;
			FOR k := MIN_VOLTAGE TO MIN(MAX_VOLTAGE,Voltage_Count)
			DO
				IF MB_NominalVoltage[k] <> 0
					AND(
					INT_TO_LREAL(MB_Voltage[k]) < INT_TO_LREAL(MB_NominalVoltage[k]) * VoltageFactor
					OR INT_TO_LREAL(MB_Voltage[k]) > INT_TO_LREAL(MB_NominalVoltage[k]) * (1.0 + (1.0 - VoltageFactor)))
				THEN
					event.no[5].Text1 						:= INT_TO_STRING(MB_Voltage[k]); 
					event.no[5].Text2 						:= INT_TO_STRING(MB_NominalVoltage[k]); 				
					event.no[5].Flag 						:= TRUE;
					EXIT;
				END_IF
			END_FOR		 
		ELSE
			event.no[5].Flag 								:= FALSE;
		END_IF
	
		event.no[6].Flag 									:= FALSE;
		event.no[7].Flag 									:= FALSE; 
		event.no[8].Flag 									:= FALSE; 
		event.no[9].Flag 									:= MAX(CPU_Temp[1],CPU_Temp[2]) > MaxTempCPU - TempWarningThreshold ; event.no[9].Text1 := INT_TO_STRING(MAX(CPU_Temp[1],CPU_Temp[2])); 
		event.no[10].Flag 									:= MB_Temp > MaxTempMB - TempWarningThreshold; event.no[10].Text1 := INT_TO_STRING(MB_Temp); 
	END_IF
	
	Event(
		ConfirmTrig	:= ConfirmTrig,
		SourceId	:= SourceId,
		no			:= ,
		Disable		:= NOT Enable,
		AutoConfirm := ,
		MIN_EVENT	=> ,
		MAX_EVENT	=> ,
		Status		=> EventStatus);
END_METHOD

END_FUNCTION_BLOCK

// POUs/IpcDiag/UPSStatus
{attribute 'no_check'}
//General UPS function block to make use of differenty types of utility power supplies 
//Requiered libs : Tc2_SUPS, Tc2_IoFunctions
FUNCTION_BLOCK UPSStatus
VAR_OUTPUT CONSTANT
	MODE_SUPS_CB3011										:	INT := 0; //SUPS for CB3011 Motherboard
	MODE_SUPS_CX50X0										:	INT := 1; //SUPS for CX50X0
	MODE_SUPS_CX51X0										:	INT := 2; //SUPS for CX51X0
	MODE_SUPS_CX9020										:	INT := 3; //SUPS for CX9020
	MODE_SUPS_BAPI											:	INT := 4; //SUPS for BAPI
	MODE_UPS_BA												:	INT := 5; //BA UPS Controller CP903x-Card (PCI/ISA) | Beckhoff P24Vxxxx USV | With Beckhoff Industrial PC's delivered APC UPS models supporting smart protocol and configured with Windows UPS Service
	MODE_UPS_EXTERN_OK										:	INT := 6; //External UPS controller connected via one Digital Input -> TRUE=PowerOK
	MODE_UPS_EXTERN_FAIL									:	INT := 7; //External UPS controller connected via one Digital Input -> TRUE=PowerFAIL
END_VAR                     								
VAR_INPUT                   													
	Enable													: 	BOOL := FALSE;		// FB will be processed as long as enable is TRUE 
	NetId													: 	T_AmsNetId 	:= '';	// AmsNet id
	Port													: 	T_AmsPort 	:= 851; // TC3 PLC RT1 = 851.... , 0 = Windows UPS service 
	Timeout													: 	TIME := DEFAULT_ADS_TIMEOUT; // Ads timeout / PowerOK/Fault delay at mode = MODE_UPS_EXTERN
	Mode													: 	INT(MODE_SUPS_CB3011..MODE_UPS_EXTERN_FAIL) := MODE_UPS_BA; // Select used UPS type
	UpsMode													: 	E_S_UPS_Mode := eSUPS_WrPersistData_Shutdown; // Used by FB_S_UPS instances and adaped for modes <> MODE_SUPS  
END_VAR
VAR_OUTPUT
	BatteryReplace											:	BOOL;
	PowerFailDetect											:	BOOL; 	//TRUE when power fail is detected 
	Status													:	E_S_UPS_State := eSUPS_PowerOK; //Reports the status of utility-supplied power into the UPS. 
	Error													:	BOOL;		//Rising edge of Error informs that an error occurred during the execution of the Function Block  	
{attribute 'displaymode':='hex'}
	ErrorID													:	UDINT; 	//Error identification 
END_VAR      
VAR              
//local *****************************************************************
	State													: 	INT := 0;
	DigInput										AT %I*	: 	BOOL; //Hardware signal for OK/NOK depending on selected UpsMode
	
//Trigger ***************************************************************

//Timer ****************************************************************
	TonPowerOff												: 	TON;	
//Instances **********************************************************  
	UPSPowerStatus											: 	FB_GetUpsStatus;
	SUPSPowerStatus_CB3011									: 	FB_S_UPS_CB3011 		:= (ePersistentMode := SPDM_2PASS);
	SUPSPowerStatus_CX50X0									: 	FB_S_UPS 				:= (iUPSPort := 16#4A8 ,ePersistentMode := SPDM_2PASS);	
	SUPSPowerStatus_CX51x0									: 	FB_S_UPS_CX51x0 		:= (iUPSPort := 16#588 ,ePersistentMode := SPDM_2PASS);
	SUPSPowerStatus_CX9020									: 	FB_S_UPS_CX9020_U900 	:= (ePersistentMode := SPDM_2PASS);
	SUPSPowerStatus_BAPI									: 	FB_S_UPS_BAPI			:= (ePersistentMode := SPDM_2PASS);
	ShutDown												: 	NT_Shutdown;
	WritePersistentData										: 	FB_WritePersistentData := (Mode := SPDM_2PASS);	
	TcStop													: 	TC_Stop;
//Dummy *****************************************************************)       								

END_VAR

	(* UPS Wrapper										*)
	(****************************************************)

(* Sequence *************************************************************************)
IF Enable THEN
	CASE state OF	
	0:
		CASE MODE OF
		MODE_SUPS_CB3011:
			SUPSPowerStatus_CB3011(
				sNetID				:= NetId,
				iPLCPort			:= Port,
				tTimeout			:= ,
				eUpsMode			:= UpsMode,
				ePersistentMode		:= ,
				tRecoverTime		:= ,
				bPowerFailDetect	=> PowerFailDetect,
				eState				=> Status);		
		
		MODE_SUPS_CX50X0:
			SUPSPowerStatus_CX50X0(
				sNetID				:= NetId,
				iPLCPort			:= Port,
				iUPSPort			:= ,
				tTimeout			:= ,
				eUpsMode			:= UpsMode,
				ePersistentMode		:= ,
				tRecoverTime		:= ,
				bPowerFailDetect	=> PowerFailDetect,
				eState				=> Status);		
			
		MODE_SUPS_CX51X0:
			SUPSPowerStatus_CX51x0(
				sNetID				:= NetId,
				iPLCPort			:= Port,
				iUPSPort			:= ,
				tTimeout			:= ,
				eUpsMode			:= UpsMode,
				ePersistentMode		:= ,
				tRecoverTime		:= ,
				bPowerFailDetect	=> PowerFailDetect,
				eState				=> Status);		
			
		MODE_SUPS_CX9020:
			SUPSPowerStatus_CX9020(
				sNetID				:= NetId,
				iPLCPort			:= Port,
				tTimeout			:= ,
				eUpsMode			:= UpsMode,
				ePersistentMode		:= ,
				tRecoverTime		:= ,
				bPowerFailDetect	=> PowerFailDetect,
				eState				=> Status);		
				
		MODE_SUPS_BAPI:
			SUPSPowerStatus_BAPI(
				sNetID				:= NetId,
				iPLCPort			:= Port,
				tTimeout			:= ,
				eUpsMode			:= UpsMode,
				ePersistentMode		:= ,
				tRecoverTime		:= ,
				bPowerFailDetect	=> PowerFailDetect,
				eState				=> Status);				

		MODE_UPS_EXTERN_OK,
		MODE_UPS_EXTERN_FAIL:
			TonPowerOff(
				IN					:= SEL(MODE = MODE_UPS_EXTERN_OK, DigInput, NOT DigInput), 
				PT					:= Timeout, 
				Q 					=> PowerFailDetect);
			Status											:= SEL(TonPowerOff.IN, eSUPS_PowerOK, eSUPS_WaitForRecover);
			IF TonPowerOff.Q                                
			THEN				                            
				Status										:= eSUPS_PowerFailure;
				state										:= 900;
			END_IF 
			
